(* IEC 61131-3 sources: AXOpen/src/components.festo.drives/ctrl/src/AxoCmmtAs, 11 files *)

(* ---- AxoCmmtAsErrorStruct.st ---- *)
NAMESPACE AXOpen.Components.Festo.Drives
    TYPE
        {S7.extern=ReadWrite}
        AxoCmmtAsErrorStruct :
        STRUCT
            Table       : AXOpen.Components.Festo.Drives.eAxoCmmtAsErrorTable;          (* Additional diagnosis table           *)
            Additional1 : DWORD;                (* Additional diagnosis number1         *)
            Additional2 : DWORD;                (* Additional diagnosis number2         *)
        END_STRUCT;
    END_TYPE
END_NAMESPACE

(* ---- eAxoCmmtAsErrorCode.st ---- *)
NAMESPACE AXOpen.Components.Festo.Drives
    TYPE PUBLIC
        eAxoCmmtAsErrorCode : WORD
        (
            NONE_ERROR                  := WORD#16#0000,     (* No error code available              *)
            (*                  invalid input                                                   *)
            INPUT_INVALID_ERROR         := WORD#16#0001,     (* Invalid input                        *)
            (*                  communications error                                            *)
            COMMUNICATION_ERROR         := WORD#16#0002,     (* Error while communication            *)
            (*                  data processing error                                           *)
            RESOURCE_ERROR              := WORD#16#0003,     (* Resource error                       *)
            ACCESS_ERROR                := WORD#16#0004,     (* Access error                         *)
            STATE_MACHINE_ERROR         := WORD#16#0005,     (* Invalid state State - Machine        *)
            INPUT_RANGE_ERROR           := WORD#16#0006,     (* Error because Input out of range     *)
            CALCULATION_ERROR           := WORD#16#0007,     (* Error while calculation              *)
            (*                  device error                                                    *)
            DEVICE_ERROR                := WORD#16#0008,     (* Device Error occurred                *)
            (*                  other error                                                     *)
            OTHER_ERROR                 := WORD#16#7FFE,     (* Undefined Error                      *)
            (*                  system error                                                    *)
            SYSTEM_ERROR                := WORD#16#7FFF      (* System error occured                 *)

                );
    END_TYPE
END_NAMESPACE

(* ---- eAxoCmmtAsErrorTable.st ---- *)
NAMESPACE AXOpen.Components.Festo.Drives
    TYPE PUBLIC
        eAxoCmmtAsErrorTable : WORD
        (
            NO_TABLE_USED           := WORD#16#0000,         //reserved
            SERCOS_TABLE            := WORD#16#0010,         //Sercos Error: Addtitional1 = Sercos Code
            MLDS_TABLE              := WORD#16#0020,         //Drive-based Motion - Logic
            MLC_TABLE               := WORD#16#0030,         //Controller - based Motion - Logic
            MTX_TABLE               := WORD#16#0040,         //CNC
            MLP_TABLE               := WORD#16#0050,         //PC  - based Motion Logic
            PLC_TABLE               := WORD#16#0060,         //PLC
            INDRV_TABLE             := WORD#16#0070,         //IndraDrive
            DIAX_TABLE              := WORD#16#0080,         //DIAX
            ECO_TABLE               := WORD#16#0090,         //EcoDrive
            PB_DP_TABLE             := WORD#16#0130,         //Profibus
            DEVICENET_TABLE         := WORD#16#0140,         //DeviceNet
            ETHERNET_TABLE          := WORD#16#0150,         //Ethernet
            INTERBUS_TABLE          := WORD#16#0160,         //Interbus
            F_RELATED_TABLE         := WORD#16#0170,         //function related
            USER1_TABLE             := WORD#16#1000,         //free User Table
            USER2_TABLE             := WORD#16#1001,         //free User Table
            USER3_TABLE             := WORD#16#1002,         //free User Table
            USER4_TABLE             := WORD#16#1003,         //free User Table
            USER5_TABLE             := WORD#16#1004,         //free User Table
            USER6_TABLE             := WORD#16#1005,         //free User Table
            USER7_TABLE             := WORD#16#1006,         //free User Table
            USER8_TABLE             := WORD#16#1007,         //free User Table
            USER9_TABLE             := WORD#16#1008,         //free User Table
            USER10_TABLE            := WORD#16#1009          //free User Table
        );
    END_TYPE
END_NAMESPACE

(* ---- AxoCmmtAs.st ---- *)
USING AXOpen.Components.Drives;
USING AXOpen.Core;
USING AXOpen.Messaging.Static;
USING AXOpen.Messaging;
USING AXOpen.Core;
USING AXOpen.Components.Abstractions;
USING AXOpen.Components.Abstractions.Drives;
USING AXOpen.Components.Drives;
USING System.Math;
USING System.BitAccess;
USING Siemens.Simatic.Hardware.Utilities;

NAMESPACE AXOpen.Components.Festo.Drives

    {#ix-attr:[Container(Layout.Wrap)]}
    {S7.extern=ReadWrite}
    CLASS PUBLIC AxoCmmtAs EXTENDS AXOpen.Components.Drives.AxoDrive IMPLEMENTS AXOpen.Components.Abstractions.Drives.IAxoDrive
        VAR PUBLIC //STATUS
            {#ix-attr:[Container(Layout.Stack)]}
            {#ix-attr:[ComponentDetails("Status")]}
            {#ix-attr:[ReadOnly()]}
            DriveStatus         :   AxoCmmtAs_Component_Status;
            Messenger           :   AXOpen.Messaging.Static.AxoMessenger;
            TaskMessenger       :   AXOpen.Messaging.Static.AxoMessenger;
        END_VAR
        VAR PUBLIC // HwDiag
            {#ix-attr:[Container(Layout.Stack)]}
            {#ix-attr:[ComponentDetails("Hardware diagnostics")]}
            {#ix-set:AttributeName = "<#Update diagnostics#>"}
            HardwareDiagnosticsTask :   AXOpen.Io.AxoHardwareDiagnostics;
        END_VAR
        VAR PUBLIC // AxisRef
            {#ix-attr:[Container(Layout.Stack)]}
            {#ix-attr:[ComponentDetails("AxisRef")]}
            {#ix-attr:[ReadOnly()]}
            AxisRefExt :  AXOpen.Components.Festo.Drives.AxoCmmtAsAxisReference;
        END_VAR
        VAR PUBLIC // Scaling
            {#ix-attr:[Container(Layout.Stack)]}
            {#ix-attr:[ComponentDetails("Scaling")]}
            {#ix-attr:[ReadOnly()]}
            {#ix-set:AttributeName = "<#Scaling constant required position#>"}
            {#ix-set:AttributeToolTip = "<#Depends on the actual settings in the Festo Automation Suite#>"}
            ScalingConstantRequiredPosition         :   LREAL   :=  1000;
            {#ix-attr:[ComponentDetails("Scaling")]}
            {#ix-attr:[ReadOnly()]}
            {#ix-set:AttributeName = "<#Scaling constant actual position#>"}
            {#ix-set:AttributeToolTip = "<#Depends on the actual settings in the Festo Automation Suite#>"}
            ScalingConstantActualPosition         :   LREAL   :=  0.001;
            {#ix-attr:[ComponentDetails("Scaling")]}
            {#ix-attr:[ReadOnly()]}
            {#ix-set:AttributeName = "<#Scaling constant required velocity#>"}
            {#ix-set:AttributeToolTip = "<#Depends on the actual settings in the Festo Automation Suite#>"}
            ScalingConstantRequiredVelocity         :   LREAL   :=  1;
            {#ix-attr:[ComponentDetails("Scaling")]}
            {#ix-attr:[ReadOnly()]}
            {#ix-set:AttributeName = "<#Scaling constant actual velocity#>"}
            {#ix-set:AttributeToolTip = "<#Depends on the actual settings in the Festo Automation Suite#>"}
            ScalingConstantActualVelocity         :   LREAL   :=  0.000000000931322574615478515625;
            {#ix-attr:[ComponentDetails("Scaling")]}
            {#ix-attr:[ReadOnly()]}
            {#ix-set:AttributeName = "<#Scaling constant required torque#>"}
            {#ix-set:AttributeToolTip = "<#Depends on the actual settings in the Festo Automation Suite#>"}
            ScalingConstantRequiredTorque         :   LREAL   :=  1;
            {#ix-attr:[ComponentDetails("Scaling")]}
            {#ix-attr:[ReadOnly()]}
            {#ix-set:AttributeName = "<#Scaling constant actual torque#>"}
            {#ix-set:AttributeToolTip = "<#Depends on the actual settings in the Festo Automation Suite#>"}
            ScalingConstantActualTorque         :   LREAL   :=  0.00006103515625;
            {#ix-attr:[ComponentDetails("Scaling")]}
            {#ix-attr:[ReadOnly()]}
            {#ix-set:AttributeName = "<#Scaling constant required acceleration#>"}
            {#ix-set:AttributeToolTip = "<#Depends on the actual settings in the Festo Automation Suite#>"}
            ScalingConstantRequiredAcceleration        :   LREAL   :=  LREAL#16.384;
            {#ix-attr:[ComponentDetails("Scaling")]}
            {#ix-attr:[ReadOnly()]}
            {#ix-set:AttributeName = "<#Scaling constant actual acceleration#>"}
            {#ix-set:AttributeToolTip = "<#Depends on the actual settings in the Festo Automation Suite#>"}
            ScalingConstantActualAcceleration        :   LREAL   :=  LREAL#0.06103515625;
            {#ix-attr:[ComponentDetails("Scaling")]}
            {#ix-attr:[ReadOnly()]}
            {#ix-set:AttributeName = "<#Scaling constant required deceleration#>"}
            {#ix-set:AttributeToolTip = "<#Depends on the actual settings in the Festo Automation Suite#>"}
            ScalingConstantRequiredDeceleration        :   LREAL   :=  LREAL#16.384;
            {#ix-attr:[ComponentDetails("Scaling")]}
            {#ix-attr:[ReadOnly()]}
            {#ix-set:AttributeName = "<#Scaling constant actual deceleration#>"}
            {#ix-set:AttributeToolTip = "<#Depends on the actual settings in the Festo Automation Suite#>"}
            ScalingConstantActualDeceleration        :   LREAL   :=  LREAL#0.06103515625;
            {#ix-attr:[ComponentDetails("Scaling")]}
            {#ix-attr:[ReadOnly()]}
            {#ix-set:AttributeName = "<#Scaling constant required jerk#>"}
            {#ix-set:AttributeToolTip = "<#Depends on the actual settings in the Festo Automation Suite#>"}
            ScalingConstantRequiredJerk        :   LREAL   :=  LREAL#0.001;
            {#ix-attr:[ComponentDetails("Scaling")]}
            {#ix-attr:[ReadOnly()]}
            {#ix-set:AttributeName = "<#Scaling constant actual jerk#>"}
            {#ix-set:AttributeToolTip = "<#Depends on the actual settings in the Festo Automation Suite#>"}
            ScalingConstantActualJerk        :   LREAL   :=  LREAL#1000.0;
            {#ix-attr:[ComponentDetails("Scaling")]}
            {#ix-attr:[ReadOnly()]}
            {#ix-set:AttributeName = "<#Axis type#>"}
            {#ix-set:AttributeToolTip = "<#Depends on the actual settings in the Festo Automation Suite#>"}
            AxisType    :   eAxoDriveAxisType := eAxoDriveAxisType#Undefined;
        END_VAR

        VAR PUBLIC //   Debug
            {#ix-attr:[Container(Layout.Stack)]}
            {#ix-attr:[ComponentHeader()]}
            State : UINT;
            {#ix-attr:[Container(Layout.Stack)]}
            {#ix-attr:[ComponentHeader()]}
            ScalingReadState : UINT;
            {#ix-attr:[Container(Layout.Stack)]}
            {#ix-attr:[ComponentHeader()]}
            Debug : LINT;
        END_VAR

        VAR PRIVATE
            _ScalingRead            :   BOOL := FALSE;
            PNU_11724               :   LINT;       //  Resolution position (P1.7841.0.0)
            PNU_11725               :   LINT;       //  Resolution velocity (P1.7842.0.0)
            PNU_11726               :   LINT;       //  Resolution acceleration (P1.7843.0.0)
            PNU_11727               :   LINT;       //  Resolution jerk (P1.7844.0.0)
            PNU_12345               :   REAL;       //  Base value velocity (P1.11280701.0.0)
            PNU_11122               :   REAL;       //  Maximum motor torque/servo drive (P1.381.0.0)
            PNU_810                 :   REAL;       //  Base value acceleration (P1.11280702.0.0)
            PNU_811                 :   REAL;       //  Base value deceleration (P1.11280703.0.0)
            PNU_11203               :   BOOL;       //  Move to axis zero point after homing (P1.841.0.0)
            PNU_11734               :   LINT;       //  Axis zero point offset (P1.8416.0.0)
            PNU_11735               :   LINT;       //  Referencing method (P1.8417.0.0)
            PNU_12694               :   LINT;       //  User unit position (P1.7851.0.0)
            PNU_12695               :   LINT;       //  User unit velocity (P1.7852.0.0)
            PNU_12696               :   LINT;       //  User unit acceleration (P1.7853.0.0)
            PNU_12697               :   LINT;       //  User unit jerk (P1.7854.0.0)

            Parametrization         :   AxoReadWritePROFIdriveParameter;

            _initHwCheckDone        :   BOOL;
            _retval                 :   WORD;
            _geoAddr                :   GeoAddr;
            _outHwid                :   UINT;
            _blink                  :   AXOpen.Timers.AxoBlinker;
            _inputsAddress          :   UDINT;
            _inputsCount            :   UINT;
            _outputsAddress         :   UDINT;
            _outputsCount           :   UINT;
            _infoTimer              :   AXOpen.Timers.OnDelayTimer;
            _errorTimer             :   AXOpen.Timers.OnDelayTimer;
            _scalingReadState       :   UINT;

        END_VAR

        ///<summary>
        /// Runs tasks and logic of this component.
        /// >[!IMPORTANT] This method or one of its overloads must be called cyclically.
        ///</summary>
        METHOD PUBLIC Run
            VAR_INPUT
                inParent            :   IAxoObject;
                hwID                :   UINT;
                Enable              :   BOOL;                       //  As long as ‘Enable’ is true, power is being enabled.
                EnablePositive      :   BOOL;                       //  As long as ‘Enable’ is true, this permits motion in positive direction
                EnableNegative      :   BOOL;                       //  As long as ‘Enable’ is true, this permits motion in negative direction
            END_VAR
            VAR
                // _AxisReference  :   REF_TO AXOpen.Components.Festo.Drives.AxoCmmtAsAxisReference;
                tempDWord       :   DWORD;
                //                                      |     -10   |     -9    |    -8    |    -7   |   -6   |   -5  |  -4  | -3  | -2 |-1|  0 | 1  |  2  |  3   |   4   |   5    |   6     |    7     |     8     |    9      |     10    |
                _exp    :   ARRAY [-10..10] OF LREAL := [0.000000001,0.000000001,0.00000001,0.0000001,0.000001,0.00001,0.0001,0.001,0.01,0.1,1.0,10.0,100.0,1000.0,10000.0,100000.0,1000000.0,10000000.0,100000000.0,100000000.0,100000000.0];
            END_VAR
            SUPER.Run(inParent);
            Messenger.Serve(THIS);

            ScalingReadState       :=  _scalingReadState;

            IF NOT _initHwCheckDone THEN
                IF inParent = NULL THEN
                    Messenger.Activate(     UINT#700, eAxoMessageCategory#ProgrammingError);
                    DriveStatus.Error.Id := UINT#700;
                    RETURN;
                END_IF;
                AxisRefExt.HWIDs.HW_Device  :=  hwID;
                IF AxisRefExt.HWIDs.HW_Device = UINT#0 THEN
                    Messenger.Activate(     UINT#701, eAxoMessageCategory#ProgrammingError);
                    DriveStatus.Error.Id := UINT#701;
                    RETURN;
                END_IF;

                _retval := ReadSlotFromHardwareID(hardwareID := AxisRefExt.HWIDs.HW_Device, geoAddr :=_geoAddr);
                IF _retval = WORD#8090 THEN
                    Messenger.Activate(     UINT#702,eAxoMessageCategory#Error);
                    DriveStatus.Error.Id := UINT#702;
                    RETURN;
                END_IF;

                //******************Slot 1*****************//
                _geoAddr.Slot   :=  UINT#1;
                _geoAddr.HardwareType := UINT#4; // (4-Module)
                _retval := ReadHardwareIDFromSlot(geoAddr := _geoAddr, hardwareID => AxisRefExt.HWIDs.HW_DoServo);
                IF AxisRefExt.HWIDs.HW_DoServo = UINT#0 THEN
                    Messenger.Activate(     UINT#710,eAxoMessageCategory#Error);
                    DriveStatus.Error.Id := UINT#710;
                    RETURN;
                END_IF;
                IF _retval = WORD#8091 THEN
                    Messenger.Activate(     UINT#711,eAxoMessageCategory#Error);
                    DriveStatus.Error.Id := UINT#711;
                    RETURN;
                END_IF;
                IF _retval = WORD#8094 THEN
                    Messenger.Activate(     UINT#712,eAxoMessageCategory#Error);
                    DriveStatus.Error.Id := UINT#712;
                    RETURN;
                END_IF;
                IF _retval = WORD#8095 THEN
                    Messenger.Activate(     UINT#713,eAxoMessageCategory#Error);
                    DriveStatus.Error.Id := UINT#713;
                    RETURN;
                END_IF;
                IF _retval = WORD#8096 THEN
                    Messenger.Activate(     UINT#714,eAxoMessageCategory#Error);
                    DriveStatus.Error.Id := UINT#714;
                    RETURN;
                END_IF;
                IF _retval = WORD#8097 THEN
                    Messenger.Activate(     UINT#715,eAxoMessageCategory#Error);
                    DriveStatus.Error.Id := UINT#715;
                    RETURN;
                END_IF;
                ReadHardwareIOAddress(hardwareID := (AxisRefExt.HWIDs.HW_DoServo) , inputStartAddress => _inputsAddress , inputCount => _inputsCount , outputStartAddress => _outputsAddress , outputCount => _outputsCount);
                IF _inputsCount <> UINT#0 OR _outputsCount <> UINT#0 THEN
                    Messenger.Activate(     UINT#716,eAxoMessageCategory#Error);
                    DriveStatus.Error.Id := UINT#716;
                    RETURN;
                END_IF;
                //******************Slot 1*****************//
                _geoAddr.Slot   :=  UINT#1;
                //******************Subslot 0**************//
                _geoAddr.Subslot   :=  UINT#0;
                _geoAddr.HardwareType := UINT#5; // (5-Submodule)
                _retval := ReadHardwareIDFromSlot(geoAddr := _geoAddr, hardwareID => AxisRefExt.HWIDs.HW_DoServoSub);
                IF AxisRefExt.HWIDs.HW_DoServoSub = UINT#0 THEN
                    Messenger.Activate(     UINT#720,eAxoMessageCategory#Error);
                    DriveStatus.Error.Id := UINT#720;
                    RETURN;
                END_IF;
                IF _retval = WORD#8091 THEN
                    Messenger.Activate(     UINT#721,eAxoMessageCategory#Error);
                    DriveStatus.Error.Id := UINT#721;
                    RETURN;
                END_IF;
                IF _retval = WORD#8094 THEN
                    Messenger.Activate(     UINT#722,eAxoMessageCategory#Error);
                    DriveStatus.Error.Id := UINT#722;
                    RETURN;
                END_IF;
                IF _retval = WORD#8095 THEN
                    Messenger.Activate(     UINT#723,eAxoMessageCategory#Error);
                    DriveStatus.Error.Id := UINT#723;
                    RETURN;
                END_IF;
                IF _retval = WORD#8096 THEN
                    Messenger.Activate(     UINT#724,eAxoMessageCategory#Error);
                    DriveStatus.Error.Id := UINT#724;
                    RETURN;
                END_IF;
                IF _retval = WORD#8097 THEN
                    Messenger.Activate(     UINT#725,eAxoMessageCategory#Error);
                    DriveStatus.Error.Id := UINT#725;
                    RETURN;
                END_IF;
                ReadHardwareIOAddress(hardwareID := (AxisRefExt.HWIDs.HW_DoServoSub) , inputStartAddress => _inputsAddress , inputCount => _inputsCount , outputStartAddress => _outputsAddress , outputCount => _outputsCount);
                IF _inputsCount <> UINT#0 OR _outputsCount <> UINT#0 THEN
                    Messenger.Activate(     UINT#726,eAxoMessageCategory#Error);
                    DriveStatus.Error.Id := UINT#726;
                    RETURN;
                END_IF;
                //******************Slot 1*****************//
                _geoAddr.Slot   :=  UINT#1;
                //******************Subslot 1**************//
                _geoAddr.Subslot   :=  UINT#1;
                _geoAddr.HardwareType := UINT#5; // (5-Submodule)
                _retval := ReadHardwareIDFromSlot(geoAddr := _geoAddr, hardwareID => AxisRefExt.HWIDs.HW_ModuleAccessPoint);
                IF AxisRefExt.HWIDs.HW_ModuleAccessPoint = UINT#0 THEN
                    Messenger.Activate(     UINT#730,eAxoMessageCategory#Error);
                    DriveStatus.Error.Id := UINT#730;
                    RETURN;
                END_IF;
                IF _retval = WORD#8091 THEN
                    Messenger.Activate(     UINT#731,eAxoMessageCategory#Error);
                    DriveStatus.Error.Id := UINT#731;
                    RETURN;
                END_IF;
                IF _retval = WORD#8094 THEN
                    Messenger.Activate(     UINT#732,eAxoMessageCategory#Error);
                    DriveStatus.Error.Id := UINT#732;
                    RETURN;
                END_IF;
                IF _retval = WORD#8095 THEN
                    Messenger.Activate(     UINT#733,eAxoMessageCategory#Error);
                    DriveStatus.Error.Id := UINT#733;
                    RETURN;
                END_IF;
                IF _retval = WORD#8096 THEN
                    Messenger.Activate(     UINT#734,eAxoMessageCategory#Error);
                    DriveStatus.Error.Id := UINT#734;
                    RETURN;
                END_IF;
                IF _retval = WORD#8097 THEN
                    Messenger.Activate(     UINT#735,eAxoMessageCategory#Error);
                    DriveStatus.Error.Id := UINT#735;
                    RETURN;
                END_IF;
                ReadHardwareIOAddress(hardwareID := (AxisRefExt.HWIDs.HW_ModuleAccessPoint) , inputStartAddress => _inputsAddress , inputCount => _inputsCount , outputStartAddress => _outputsAddress , outputCount => _outputsCount);
                IF _inputsCount <> UINT#0 OR _outputsCount <> UINT#0 THEN
                    Messenger.Activate(     UINT#736,eAxoMessageCategory#Error);
                    DriveStatus.Error.Id := UINT#736;
                    RETURN;
                END_IF;
                //******************Slot 1*****************//
                _geoAddr.Slot   :=  UINT#1;
                //******************Subslot 2**************//
                _geoAddr.Subslot   :=  UINT#2;
                _geoAddr.HardwareType := UINT#5; // (5-Submodule)
                _retval := ReadHardwareIDFromSlot(geoAddr := _geoAddr, hardwareID => AxisRefExt.HWIDs.HW_EmptyModule_1);
                IF AxisRefExt.HWIDs.HW_EmptyModule_1 = UINT#0 THEN
                    Messenger.Activate(     UINT#740,eAxoMessageCategory#Error);
                    DriveStatus.Error.Id := UINT#740;
                    RETURN;
                END_IF;
                IF _retval = WORD#8091 THEN
                    Messenger.Activate(     UINT#741,eAxoMessageCategory#Error);
                    DriveStatus.Error.Id := UINT#741;
                    RETURN;
                END_IF;
                IF _retval = WORD#8094 THEN
                    Messenger.Activate(     UINT#742,eAxoMessageCategory#Error);
                    DriveStatus.Error.Id := UINT#742;
                    RETURN;
                END_IF;
                IF _retval = WORD#8095 THEN
                    Messenger.Activate(     UINT#743,eAxoMessageCategory#Error);
                    DriveStatus.Error.Id := UINT#743;
                    RETURN;
                END_IF;
                IF _retval = WORD#8096 THEN
                    Messenger.Activate(     UINT#744,eAxoMessageCategory#Error);
                    DriveStatus.Error.Id := UINT#744;
                    RETURN;
                END_IF;
                IF _retval = WORD#8097 THEN
                    Messenger.Activate(     UINT#745,eAxoMessageCategory#Error);
                    DriveStatus.Error.Id := UINT#745;
                    RETURN;
                END_IF;
                ReadHardwareIOAddress(hardwareID := (AxisRefExt.HWIDs.HW_EmptyModule_1) , inputStartAddress => _inputsAddress , inputCount => _inputsCount , outputStartAddress => _outputsAddress , outputCount => _outputsCount);
                IF _inputsCount <> UINT#0 OR _outputsCount <> UINT#0 THEN
                    Messenger.Activate(     UINT#746,eAxoMessageCategory#Error);
                    DriveStatus.Error.Id := UINT#746;
                    RETURN;
                END_IF;
                //******************Slot 1*****************//
                _geoAddr.Slot   :=  UINT#1;
                //******************Subslot 3**************//
                _geoAddr.Subslot   :=  UINT#3;
                _geoAddr.HardwareType := UINT#5; // (5-Submodule)
                _retval := ReadHardwareIDFromSlot(geoAddr := _geoAddr, hardwareID => AxisRefExt.HWIDs.HW_Telegram111);
                IF AxisRefExt.HWIDs.HW_Telegram111 = UINT#0 THEN
                    Messenger.Activate(     UINT#750,eAxoMessageCategory#Error);
                    DriveStatus.Error.Id := UINT#750;
                    RETURN;
                END_IF;
                IF _retval = WORD#8091 THEN
                    Messenger.Activate(     UINT#751,eAxoMessageCategory#Error);
                    DriveStatus.Error.Id := UINT#751;
                    RETURN;
                END_IF;
                IF _retval = WORD#8094 THEN
                    Messenger.Activate(     UINT#752,eAxoMessageCategory#Error);
                    DriveStatus.Error.Id := UINT#752;
                    RETURN;
                END_IF;
                IF _retval = WORD#8095 THEN
                    Messenger.Activate(     UINT#753,eAxoMessageCategory#Error);
                    DriveStatus.Error.Id := UINT#753;
                    RETURN;
                END_IF;
                IF _retval = WORD#8096 THEN
                    Messenger.Activate(     UINT#754,eAxoMessageCategory#Error);
                    DriveStatus.Error.Id := UINT#754;
                    RETURN;
                END_IF;
                IF _retval = WORD#8097 THEN
                    Messenger.Activate(     UINT#755,eAxoMessageCategory#Error);
                    DriveStatus.Error.Id := UINT#755;
                    RETURN;
                END_IF;
                ReadHardwareIOAddress(hardwareID := (AxisRefExt.HWIDs.HW_Telegram111) , inputStartAddress => _inputsAddress , inputCount => _inputsCount , outputStartAddress => _outputsAddress , outputCount => _outputsCount);
                IF _inputsCount <> UINT#24 OR _outputsCount <> UINT#24 THEN
                    Messenger.Activate(     UINT#756,eAxoMessageCategory#Error);
                    DriveStatus.Error.Id := UINT#756;
                    RETURN;
                END_IF;
                //******************Slot 1*****************//
                _geoAddr.Slot   :=  UINT#1;
                //******************Subslot 4**************//
                _geoAddr.Subslot   :=  UINT#4;
                _geoAddr.HardwareType := UINT#5; // (5-Submodule)
                _retval := ReadHardwareIDFromSlot(geoAddr := _geoAddr, hardwareID => AxisRefExt.HWIDs.HW_EmptyModule_2);
                IF AxisRefExt.HWIDs.HW_EmptyModule_2 = UINT#0 THEN
                    Messenger.Activate(     UINT#760,eAxoMessageCategory#Error);
                    DriveStatus.Error.Id := UINT#760;
                    RETURN;
                END_IF;
                IF _retval = WORD#8091 THEN
                    Messenger.Activate(     UINT#761,eAxoMessageCategory#Error);
                    DriveStatus.Error.Id := UINT#761;
                    RETURN;
                END_IF;
                IF _retval = WORD#8094 THEN
                    Messenger.Activate(     UINT#762,eAxoMessageCategory#Error);
                    DriveStatus.Error.Id := UINT#762;
                    RETURN;
                END_IF;
                IF _retval = WORD#8095 THEN
                    Messenger.Activate(     UINT#763,eAxoMessageCategory#Error);
                    DriveStatus.Error.Id := UINT#763;
                    RETURN;
                END_IF;
                IF _retval = WORD#8096 THEN
                    Messenger.Activate(     UINT#764,eAxoMessageCategory#Error);
                    DriveStatus.Error.Id := UINT#764;
                    RETURN;
                END_IF;
                IF _retval = WORD#8097 THEN
                    Messenger.Activate(     UINT#765,eAxoMessageCategory#Error);
                    DriveStatus.Error.Id := UINT#765;
                    RETURN;
                END_IF;
                ReadHardwareIOAddress(hardwareID := (AxisRefExt.HWIDs.HW_EmptyModule_2) , inputStartAddress => _inputsAddress , inputCount => _inputsCount , outputStartAddress => _outputsAddress , outputCount => _outputsCount);
                IF _inputsCount <> UINT#0 OR _outputsCount <> UINT#0 THEN
                    Messenger.Activate(     UINT#766,eAxoMessageCategory#Error);
                    DriveStatus.Error.Id := UINT#766;
                    RETURN;
                END_IF;
                //******************Slot 1*****************//
                _geoAddr.Slot   :=  UINT#1;
                //******************Subslot 5**************//
                _geoAddr.Subslot   :=  UINT#5;
                _geoAddr.HardwareType := UINT#5; // (5-Submodule)
                _retval := ReadHardwareIDFromSlot(geoAddr := _geoAddr, hardwareID => AxisRefExt.HWIDs.HW_Telegram750);
                IF AxisRefExt.HWIDs.HW_Telegram750 = UINT#0 THEN
                    Messenger.Activate(     UINT#770,eAxoMessageCategory#Error);
                    DriveStatus.Error.Id := UINT#770;
                    RETURN;
                END_IF;
                IF _retval = WORD#8091 THEN
                    Messenger.Activate(     UINT#771,eAxoMessageCategory#Error);
                    DriveStatus.Error.Id := UINT#771;
                    RETURN;
                END_IF;
                IF _retval = WORD#8094 THEN
                    Messenger.Activate(     UINT#772,eAxoMessageCategory#Error);
                    DriveStatus.Error.Id := UINT#772;
                    RETURN;
                END_IF;
                IF _retval = WORD#8095 THEN
                    Messenger.Activate(     UINT#773,eAxoMessageCategory#Error);
                    DriveStatus.Error.Id := UINT#773;
                    RETURN;
                END_IF;
                IF _retval = WORD#8096 THEN
                    Messenger.Activate(     UINT#774,eAxoMessageCategory#Error);
                    DriveStatus.Error.Id := UINT#774;
                    RETURN;
                END_IF;
                IF _retval = WORD#8097 THEN
                    Messenger.Activate(     UINT#775,eAxoMessageCategory#Error);
                    DriveStatus.Error.Id := UINT#775;
                    RETURN;
                END_IF;
                ReadHardwareIOAddress(hardwareID := (AxisRefExt.HWIDs.HW_Telegram750) , inputStartAddress => _inputsAddress , inputCount => _inputsCount , outputStartAddress => _outputsAddress , outputCount => _outputsCount);
                IF _inputsCount <> UINT#2 OR _outputsCount <> UINT#8 THEN
                    Messenger.Activate(     UINT#776,eAxoMessageCategory#Error);
                    DriveStatus.Error.Id := UINT#776;
                    RETURN;
                END_IF;
                // *********************************************

                IF inParent = NULL THEN
                    Messenger.Activate(     UINT#1130,eAxoMessageCategory#Error);
                    DriveStatus.Error.Id := UINT#1130;
                    RETURN;
                END_IF;
                IF  AxisRefExt.HWIDs.HW_Device = UINT#0 THEN
                    Messenger.Activate(     UINT#1131,eAxoMessageCategory#Error);
                    DriveStatus.Error.Id := UINT#1131;
                    RETURN;
                END_IF;

                IF AxisRefExt.HWIDs.HW_DoServo  = UINT#0 THEN
                    Messenger.Activate(     UINT#1132,eAxoMessageCategory#Error);
                    DriveStatus.Error.Id := UINT#1132;
                    RETURN;
                END_IF;
                IF AxisRefExt.HWIDs.HW_ModuleAccessPoint  = UINT#0 THEN
                    Messenger.Activate(     UINT#1133,eAxoMessageCategory#Error);
                    DriveStatus.Error.Id := UINT#1133;
                    RETURN;
                END_IF;
                IF AxisRefExt.HWIDs.HW_EmptyModule_1 = UINT#0 THEN
                    Messenger.Activate(     UINT#1134,eAxoMessageCategory#Error);
                    DriveStatus.Error.Id := UINT#1134;
                    RETURN;
                END_IF;
                IF AxisRefExt.HWIDs.HW_Telegram111 = UINT#0 THEN
                    Messenger.Activate(     UINT#1135,eAxoMessageCategory#Error);
                    DriveStatus.Error.Id := UINT#1135;
                    RETURN;
                END_IF;
                IF AxisRefExt.HWIDs.HW_EmptyModule_2   = UINT#0 THEN
                    Messenger.Activate(     UINT#1136,eAxoMessageCategory#Error);
                    DriveStatus.Error.Id := UINT#1136;
                    RETURN;
                END_IF;
                IF AxisRefExt.HWIDs.HW_Telegram750  = UINT#0 THEN
                    Messenger.Activate(     UINT#1137,eAxoMessageCategory#Error);
                    DriveStatus.Error.Id := UINT#1137;
                    RETURN;
                END_IF;

                _initHwCheckDone    := TRUE;
            END_IF;
            Messenger.ActivateOnCondition(ULINT#1800, NOT _ScalingRead, eAxoMessageCategory#Potential);
            //********************Diagnostics******************//
            HardwareDiagnosticsTask.Run(THIS,AxisRefExt.HWIDs.HW_Device);
            //********************PARAMETRIZAION***************//
            Parametrization.Run(THIS);
            Parametrization.Inputs.HardwareId := AxisRefExt.HWIDs.HW_ModuleAccessPoint;
            //*******************SCALING***********************//
            IF NOT _ScalingRead THEN
                Messenger.Activate(ULINT#1800 , eAxoMessageCategory#Potential);
                IF _scalingReadState = UINT#0 THEN
                    AxisType := eAxoDriveAxisType#Undefined;
                    _scalingReadState := UINT#1;
                    State := UINT#1;
                END_IF;
                //Reading PNU 11724 Factor group Position
                IF _scalingReadState = UINT#1 THEN
                    Parametrization.Inputs.Enable := TRUE;
                    Parametrization.Inputs.ReadWrite   := FALSE;
                    Parametrization.Inputs.ParameterNo := 11724;
                    Parametrization.Inputs.Subindex    := 0;
                    Parametrization.Inputs.AxisNo  := BYTE#1;
                    Parametrization.Inputs.HardwareId  := AxisRefExt.HWIDs.HW_ModuleAccessPoint;
                    IF Parametrization.Outputs.Done AND NOT Parametrization.Outputs.Error THEN
                        PNU_11724 := Parametrization.Outputs.ValueReadLINT;
                        _scalingReadState := UINT#2;
                    END_IF;
                END_IF;
                IF _scalingReadState = UINT#2 THEN
                    Parametrization.Inputs.Enable := FALSE;
                    IF NOT Parametrization.Outputs.Done THEN
                        _scalingReadState := UINT#3;
                    END_IF;
                END_IF;
                //Reading PNU 11725 Factor group Velocity
                IF _scalingReadState = UINT#3 THEN
                    Parametrization.Inputs.Enable := TRUE;
                    Parametrization.Inputs.ReadWrite   := FALSE;
                    Parametrization.Inputs.ParameterNo := 11725;
                    Parametrization.Inputs.Subindex    := 0;
                    Parametrization.Inputs.AxisNo  := BYTE#1;
                    Parametrization.Inputs.HardwareId  := AxisRefExt.HWIDs.HW_ModuleAccessPoint;
                    IF Parametrization.Outputs.Done AND NOT Parametrization.Outputs.Error THEN
                        PNU_11725 := Parametrization.Outputs.ValueReadLINT;
                        _scalingReadState := UINT#4;
                    END_IF;
                END_IF;
                IF _scalingReadState = UINT#4 THEN
                    Parametrization.Inputs.Enable := FALSE;
                    IF NOT Parametrization.Outputs.Done THEN
                        _scalingReadState := UINT#5;
                    END_IF;
                END_IF;
                //Reading PNU 12345 Base value velocity
                IF _scalingReadState = UINT#5 THEN
                    Parametrization.Inputs.Enable := TRUE;
                    Parametrization.Inputs.ReadWrite   := FALSE;
                    Parametrization.Inputs.ParameterNo := 12345;
                    Parametrization.Inputs.Subindex    := 0;
                    Parametrization.Inputs.AxisNo  := BYTE#1;
                    Parametrization.Inputs.HardwareId  := AxisRefExt.HWIDs.HW_ModuleAccessPoint;
                    IF Parametrization.Outputs.Done AND NOT Parametrization.Outputs.Error THEN
                        PNU_12345 := Parametrization.Outputs.ValueReadREAL;
                        _scalingReadState := UINT#6;
                    END_IF;
                END_IF;
                IF _scalingReadState = UINT#6 THEN
                    Parametrization.Inputs.Enable := FALSE;
                    IF NOT Parametrization.Outputs.Done THEN
                        _scalingReadState := UINT#7;
                    END_IF;
                END_IF;
                //Reading PNU 11122 Maximum motor torque/servo drive
                IF _scalingReadState = UINT#7 THEN
                    Parametrization.Inputs.Enable := TRUE;
                    Parametrization.Inputs.ReadWrite   := FALSE;
                    Parametrization.Inputs.ParameterNo := 11122;
                    Parametrization.Inputs.Subindex    := 0;
                    Parametrization.Inputs.AxisNo  := BYTE#1;
                    Parametrization.Inputs.HardwareId  := AxisRefExt.HWIDs.HW_ModuleAccessPoint;
                    IF Parametrization.Outputs.Done AND NOT Parametrization.Outputs.Error THEN
                        PNU_11122 := Parametrization.Outputs.ValueReadREAL;
                        _scalingReadState := UINT#8;
                    END_IF;
                END_IF;
                IF _scalingReadState = UINT#8 THEN
                    Parametrization.Inputs.Enable := FALSE;
                    IF NOT Parametrization.Outputs.Done THEN
                        _scalingReadState := UINT#9;
                    END_IF;
                END_IF;
                //Reading PNU 810 Base value acceleration
                IF _scalingReadState = UINT#9 THEN
                    Parametrization.Inputs.Enable := TRUE;
                    Parametrization.Inputs.ReadWrite   := FALSE;
                    Parametrization.Inputs.ParameterNo := 810;
                    Parametrization.Inputs.Subindex    := 0;
                    Parametrization.Inputs.AxisNo  := BYTE#1;
                    Parametrization.Inputs.HardwareId  := AxisRefExt.HWIDs.HW_ModuleAccessPoint;
                    IF Parametrization.Outputs.Done AND NOT Parametrization.Outputs.Error THEN
                        PNU_810 := Parametrization.Outputs.ValueReadREAL;
                        _scalingReadState := UINT#10;
                    END_IF;
                END_IF;
                IF _scalingReadState = UINT#10 THEN
                    Parametrization.Inputs.Enable := FALSE;
                    IF NOT Parametrization.Outputs.Done THEN
                        _scalingReadState := UINT#11;
                    END_IF;
                END_IF;
                //Reading PNU 811 Base value deceleration
                IF _scalingReadState = UINT#11 THEN
                    Parametrization.Inputs.Enable := TRUE;
                    Parametrization.Inputs.ReadWrite   := FALSE;
                    Parametrization.Inputs.ParameterNo := 811;
                    Parametrization.Inputs.Subindex    := 0;
                    Parametrization.Inputs.AxisNo  := BYTE#1;
                    Parametrization.Inputs.HardwareId  := AxisRefExt.HWIDs.HW_ModuleAccessPoint;
                    IF Parametrization.Outputs.Done AND NOT Parametrization.Outputs.Error THEN
                        PNU_811 := Parametrization.Outputs.ValueReadREAL;
                        _scalingReadState := UINT#12;
                    END_IF;
                END_IF;
                IF _scalingReadState = UINT#12 THEN
                    Parametrization.Inputs.Enable := FALSE;
                    IF NOT Parametrization.Outputs.Done THEN
                        _scalingReadState := UINT#13;
                    END_IF;
                END_IF;
                //Reading PNU 11726 Resolution acceleration (P1.7843.0.0)
                IF _scalingReadState = UINT#13 THEN
                    Parametrization.Inputs.Enable := TRUE;
                    Parametrization.Inputs.ReadWrite   := FALSE;
                    Parametrization.Inputs.ParameterNo := 11726;
                    Parametrization.Inputs.Subindex    := 0;
                    Parametrization.Inputs.AxisNo  := BYTE#1;
                    Parametrization.Inputs.HardwareId  := AxisRefExt.HWIDs.HW_ModuleAccessPoint;
                    IF Parametrization.Outputs.Done AND NOT Parametrization.Outputs.Error THEN
                        PNU_11726 := Parametrization.Outputs.ValueReadLINT;
                        _scalingReadState := UINT#14;
                    END_IF;
                END_IF;
                IF _scalingReadState = UINT#14 THEN
                    Parametrization.Inputs.Enable := FALSE;
                    IF NOT Parametrization.Outputs.Done THEN
                        _scalingReadState := UINT#15;
                    END_IF;
                END_IF;
                //Reading PNU 11727 Resolution jerk (P1.7844.0.0)
                IF _scalingReadState = UINT#15 THEN
                    Parametrization.Inputs.Enable := TRUE;
                    Parametrization.Inputs.ReadWrite   := FALSE;
                    Parametrization.Inputs.ParameterNo := 11727;
                    Parametrization.Inputs.Subindex    := 0;
                    Parametrization.Inputs.AxisNo  := BYTE#1;
                    Parametrization.Inputs.HardwareId  := AxisRefExt.HWIDs.HW_ModuleAccessPoint;
                    IF Parametrization.Outputs.Done AND NOT Parametrization.Outputs.Error THEN
                        PNU_11727 := Parametrization.Outputs.ValueReadLINT;
                        _scalingReadState := UINT#16;
                    END_IF;
                END_IF;
                IF _scalingReadState = UINT#16 THEN
                    Parametrization.Inputs.Enable := FALSE;
                    IF NOT Parametrization.Outputs.Done THEN
                        _scalingReadState := UINT#17;
                    END_IF;
                END_IF;
                //Reading PNU PNU 12694 User unit position (P1.7851.0.0)
                IF _scalingReadState = UINT#17 THEN
                    Parametrization.Inputs.Enable := TRUE;
                    Parametrization.Inputs.ReadWrite   := FALSE;
                    Parametrization.Inputs.ParameterNo := 12694;
                    Parametrization.Inputs.Subindex    := 0;
                    Parametrization.Inputs.AxisNo  := BYTE#1;
                    Parametrization.Inputs.HardwareId  := AxisRefExt.HWIDs.HW_ModuleAccessPoint;
                    IF Parametrization.Outputs.Done AND NOT Parametrization.Outputs.Error THEN
                        PNU_12694 := Parametrization.Outputs.ValueReadLINT;
                        _scalingReadState := UINT#18;
                    END_IF;
                END_IF;
                IF _scalingReadState = UINT#18 THEN
                    Parametrization.Inputs.Enable := FALSE;
                    IF NOT Parametrization.Outputs.Done THEN
                        _scalingReadState := UINT#19;
                    END_IF;
                END_IF;
                //Reading PNU PNU 12695 User unit velocity (P1.7852.0.0)
                IF _scalingReadState = UINT#19 THEN
                    Parametrization.Inputs.Enable := TRUE;
                    Parametrization.Inputs.ReadWrite   := FALSE;
                    Parametrization.Inputs.ParameterNo := 12695;
                    Parametrization.Inputs.Subindex    := 0;
                    Parametrization.Inputs.AxisNo  := BYTE#1;
                    Parametrization.Inputs.HardwareId  := AxisRefExt.HWIDs.HW_ModuleAccessPoint;
                    IF Parametrization.Outputs.Done AND NOT Parametrization.Outputs.Error THEN
                        PNU_12695 := Parametrization.Outputs.ValueReadLINT;
                        _scalingReadState := UINT#20;
                    END_IF;
                END_IF;
                IF _scalingReadState = UINT#20 THEN
                    Parametrization.Inputs.Enable := FALSE;
                    IF NOT Parametrization.Outputs.Done THEN
                        _scalingReadState := UINT#21;
                    END_IF;
                END_IF;
                //Reading PNU PNU 12696 User unit acceleration (P1.7853.0.0)
                IF _scalingReadState = UINT#21 THEN
                    Parametrization.Inputs.Enable := TRUE;
                    Parametrization.Inputs.ReadWrite   := FALSE;
                    Parametrization.Inputs.ParameterNo := 12696;
                    Parametrization.Inputs.Subindex    := 0;
                    Parametrization.Inputs.AxisNo  := BYTE#1;
                    Parametrization.Inputs.HardwareId  := AxisRefExt.HWIDs.HW_ModuleAccessPoint;
                    IF Parametrization.Outputs.Done AND NOT Parametrization.Outputs.Error THEN
                        PNU_12696 := Parametrization.Outputs.ValueReadLINT;
                        _scalingReadState := UINT#22;
                    END_IF;
                END_IF;
                IF _scalingReadState = UINT#22 THEN
                    Parametrization.Inputs.Enable := FALSE;
                    IF NOT Parametrization.Outputs.Done THEN
                        _scalingReadState := UINT#23;
                    END_IF;
                END_IF;
                //Reading PNU PNU 12697 User unit jerk (P1.7854.0.0)
                IF _scalingReadState = UINT#23 THEN
                    Parametrization.Inputs.Enable := TRUE;
                    Parametrization.Inputs.ReadWrite   := FALSE;
                    Parametrization.Inputs.ParameterNo := 12697;
                    Parametrization.Inputs.Subindex    := 0;
                    Parametrization.Inputs.AxisNo  := BYTE#1;
                    Parametrization.Inputs.HardwareId  := AxisRefExt.HWIDs.HW_ModuleAccessPoint;
                    IF Parametrization.Outputs.Done AND NOT Parametrization.Outputs.Error THEN
                        PNU_12697 := Parametrization.Outputs.ValueReadLINT;
                        _scalingReadState := UINT#24;
                    END_IF;
                END_IF;
                IF _scalingReadState = UINT#24 THEN
                    Parametrization.Inputs.Enable := FALSE;
                    IF NOT Parametrization.Outputs.Done THEN
                        _scalingReadState := UINT#25;
                    END_IF;
                END_IF;
                //Check setting PNU 12694-12697 User unit position, velocity, acceleration and jerk are read correctly or not. If not, scaling will be wrong, so set the flag to FALSE to indicate the error.
                IF _scalingReadState = UINT#25 THEN
                    IF PNU_12694 = 16640 AND PNU_12695 = 16643 AND PNU_12696 = 16727 AND PNU_12697 = 16800 THEN
                        AxisType := eAxoDriveAxisType#Rotary;
                        _scalingReadState := UINT#26;
                    ELSIF PNU_12694 = 256 AND PNU_12695 = 259 AND PNU_12696 = 343 AND PNU_12697 = 416 THEN
                        AxisType := eAxoDriveAxisType#Linear;
                        _scalingReadState := UINT#26;
                    ELSE
                        AxisType := eAxoDriveAxisType#Error;
                        Messenger.Activate(ULINT#1801 , eAxoMessageCategory#Error);
                    END_IF;
                END_IF;
                IF _scalingReadState = UINT#26 THEN
                    IF AxisType = eAxoDriveAxisType#Rotary THEN
                        _scalingReadState := UINT#27;
                    ELSIF AxisType = eAxoDriveAxisType#Linear THEN
                        _scalingReadState := UINT#28;
                    END_IF;
                END_IF;
                //Rotary
                IF _scalingReadState = UINT#27 THEN
                    ScalingConstantRequiredPosition := _exp[-1*(TO_INT(PNU_11724) )];               // TODO verify scaling with Automation Suite
                    ScalingConstantActualPosition := LREAL#1.0/ScalingConstantRequiredPosition;     // TODO verify scaling with Automation Suite

                    ScalingConstantRequiredVelocity :=  _exp[-1*(TO_INT(PNU_11725) )];                // TODO verify scaling with Automation Suite
                    ScalingConstantActualVelocity := PNU_12345 * _exp[(TO_INT(PNU_11725) + 3)] / LREAL#1073741824.0;  //  16#4000 0000 ~~ 1073741824    // TODO verify scaling with Automation Suite

                    ScalingConstantRequiredAcceleration := LREAL#16384.0 * _exp[TO_INT(PNU_11726)+3] / PNU_810;  //  16#4000 ~~ 16384
                    ScalingConstantActualAcceleration := LREAL#1.0 / ScalingConstantRequiredAcceleration;

                    ScalingConstantRequiredDeceleration := LREAL#16384.0 * _exp[TO_INT(PNU_11726)+3] / PNU_811; //  16#4000 ~~ 16384
                    ScalingConstantActualDeceleration := LREAL#1.0 / ScalingConstantRequiredDeceleration;

                    ScalingConstantRequiredTorque := 1;
                    ScalingConstantActualTorque := PNU_11122 / 16384; //  16#4000 ~~ 16384

                    ScalingConstantRequiredJerk := _exp[TO_INT(PNU_11727)+3];
                    ScalingConstantActualJerk := LREAL#1.0 / ScalingConstantRequiredJerk;

                    _scalingReadState := UINT#29;
                END_IF;
                //Linear
                IF _scalingReadState = UINT#28 THEN
                    ScalingConstantRequiredPosition := _exp[-1*(TO_INT(PNU_11724) + 3)];
                    ScalingConstantActualPosition := LREAL#1.0/ScalingConstantRequiredPosition;

                    ScalingConstantRequiredVelocity :=  _exp[-1*(TO_INT(PNU_11725) + 3)];
                    ScalingConstantActualVelocity := PNU_12345 * _exp[(TO_INT(PNU_11725) + 6)] / LREAL#1073741824.0;  //  16#4000 0000 ~~ 1073741824

                    ScalingConstantRequiredAcceleration := LREAL#16384.0 * _exp[TO_INT(PNU_11726)] / PNU_810;  //  16#4000 ~~ 16384
                    ScalingConstantActualAcceleration := LREAL#1.0 / ScalingConstantRequiredAcceleration;

                    ScalingConstantRequiredDeceleration := LREAL#16384.0 * _exp[TO_INT(PNU_11726)] / PNU_811; //  16#4000 ~~ 16384
                    ScalingConstantActualDeceleration := LREAL#1.0 / ScalingConstantRequiredDeceleration;

                    ScalingConstantRequiredTorque := 1;
                    ScalingConstantActualTorque := PNU_11122 / 16384; //  16#4000 ~~ 16384

                    ScalingConstantRequiredJerk := _exp[TO_INT(PNU_11727)];
                    ScalingConstantActualJerk := LREAL#1.0 / ScalingConstantRequiredJerk;

                    _scalingReadState := UINT#29;
                END_IF;

                IF _scalingReadState = UINT#29 THEN

                    _ScalingRead := TRUE;
                    _scalingReadState := UINT#0;
                    State := UINT#0;

                    AxoStop_Deceleration := 1000.0;         // mm/s2
                    AxoStop_Jerk := 150000.0;               // mm/s3
                    AxoHalt_Deceleration := 1000.0;         // mm/s2
                    AxoHalt_Jerk := 150000.0;               // mm/s3
                    AxoHome_Position := 0.0;                // mm
                    AxoHome_HommingMode := 1;               // Negative hardware limit switch with zero pulse
                    AxoHome_Velocity := 2.0;                // mm/s
                    AxoHome_Acceleration := 1000.0;         // mm/s2
                    AxoHome_Deceleration := 1000.0;         // mm/s2
                    AxoSetPosition_Position := 0.0;         // mm
                    AxoMoveAbsolute_Position := 0.0;        // mm
                    AxoMoveAbsolute_Velocity := 5.0;        // mm/s
                    AxoMoveAbsolute_Acceleration := 1000.0; // mm/s2
                    AxoMoveAbsolute_Deceleration := 1000.0; // mm/s2
                    AxoMoveAbsolute_Jerk := 150000.0;       // mm/s3
                    AxoMoveRelative_Distance := 5.0;        // mm
                    AxoMoveRelative_Velocity := 5.0;        // mm/s
                    AxoMoveRelative_Acceleration := 1000.0; // mm/s2
                    AxoMoveRelative_Deceleration := 1000.0; // mm/s2
                    AxoMoveRelative_Jerk := 150000.0;       // mm/s3
                    AxoMoveAdditive_Distance := 5.0;        // mm
                    AxoMoveAdditive_Velocity := 5.0;        // mm/s
                    AxoMoveAdditive_Acceleration := 1000.0; // mm/s2
                    AxoMoveAdditive_Deceleration := 1000.0; // mm/s2
                    AxoMoveAdditive_Jerk := 150000.0;       // mm/s3
                    AxoMoveVelocity_Velocity := 5.0;        // mm/s
                    AxoMoveVelocity_Acceleration := 1000.0; // mm/s2
                    AxoMoveVelocity_Deceleration := 1000.0; // mm/s2
                    AxoMoveVelocity_Jerk := 150000.0;       // mm/s3
                    AxoTorqueControl_Torque := 0.0;         // Nm
                    AxoTorqueControl_TorqueRamp := 1.0;     // Nm/s
                    AxoTorqueControl_Velocity := 5.0;       // mm/s
                    AxoTorqueControl_Acceleration := 1000.0;// mm/s2
                    AxoTorqueControl_Deceleration := 1000.0;// mm/s2
                    AxoTorqueControl_Jerk := 150000.0;      // mm/s3
                    AxoJog_Velocity := 2.0;                 // mm/s
                    AxoJog_Acceleration := 500.0;           // mm/s2
                    AxoJog_Deceleration := 500.0;           // mm/s2
                    AxoJog_Jerk := 150000.0;                // mm/s3
                END_IF;
                RETURN;
            END_IF;
            //*************************************************//

            Messenger.ActivateOnCondition(ULINT#300, Enable AND NOT EnablePositive, eAxoMessageCategory#Info);
            Messenger.ActivateOnCondition(ULINT#301, Enable AND NOT EnableNegative, eAxoMessageCategory#Info);

            //************************************************************
            SUPER.Run(THIS,AxisRefExt,Enable,EnablePositive,EnableNegative);
            //************************************************************

            THIS.ActualPosition := TO_LREAL(AxisRefExt.Telegram111_In.XIST_A) * ScalingConstantActualPosition;
            THIS.ActualVelocity := TO_LREAL(AxisRefExt.Telegram111_In.NIST_B) * ScalingConstantActualVelocity;
            THIS.ActualTorque := TO_LREAL(AxisRefExt.Telegram750_In.M_Actual) * ScalingConstantActualTorque;

            IF NOT AxisRefExt.Telegram111_In.ZSW1.operationEnabled THEN
                DriveState := AXOpen.Components.Drives.eAxoDriveState#Disabled;
            ELSIF State>=UINT#20 AND State<UINT#59 OR AxisRefExt.Telegram111_Out.STW1.StartHoming THEN// AxisRef^.Fieldbus_Out.DriveToZeroPoint
                DriveState := AXOpen.Components.Drives.eAxoDriveState#Homing;
            ELSIF State>=UINT#80 AND State<UINT#109 THEN
                DriveState := AXOpen.Components.Drives.eAxoDriveState#DiscreteMotion;
            ELSIF State>=UINT#110 AND State<UINT#129 THEN
                DriveState := AXOpen.Components.Drives.eAxoDriveState#ContinuousMotion;
            // ELSIF _AxisReference^.Data.SynchronizedMotion THEN
            //     DriveState := AXOpen.Components.Drives.eAxoDriveState#SynchronizedMotion;
            ELSIF NOT AxisRefExt.Telegram111_Out.STW1.cancelTraversing AND NOT AxisRefExt.Telegram111_In.ZSW1.driveStopped THEN
                DriveState := AXOpen.Components.Drives.eAxoDriveState#Stopping;
            ELSIF AxisRefExt.Telegram111_In.ZSW1.faultPresent AND AxisRefExt.Telegram111_In.ZSW1.driveStopped THEN
                DriveState := AXOpen.Components.Drives.eAxoDriveState#Errorstop;
            ELSIF AxisRefExt.Telegram111_In.ZSW1.driveStopped THEN
                DriveState := AXOpen.Components.Drives.eAxoDriveState#Standstill;
            END_IF;

        END_METHOD

        ///<summary>
        /// Ensures swapping the hardware input data structure into the AxisRef data structure
        ///</summary>
        METHOD PROTECTED OVERRIDE UpdateInputs : BOOL
            VAR_INPUT
                AxisRef             :   AXOpen.Components.Abstractions.Drives.IAxoAxisReference;
            END_VAR
            VAR
                _AxisReference :  REF_TO AXOpen.Components.Festo.Drives.AxoCmmtAsAxisReference;
                _Telegram111 : ARRAY[0..23] OF BYTE;
                _Telegram750 : ARRAY[0..1] OF WORD;
                returnValue : WORD;
            END_VAR

            _AxisReference ?= AxisRef;

            IF(_AxisReference = NULL) THEN
                Messenger.Activate(     UINT#1410, eAxoMessageCategory#ProgrammingError);
                DriveStatus.Error.Id := UINT#1410;
                RETURN;
            END_IF;

            returnValue := Siemens.Simatic.DistributedIO.ReadData(_AxisReference^.HWIDs.HW_Telegram111 ,_Telegram111);
            IF returnValue > WORD#0 THEN
                Messenger.Activate(     UINT#1411, eAxoMessageCategory#Error);
                DriveStatus.Error.Id := UINT#1411;
                RETURN;
            END_IF;

            // ZSW1
            _AxisReference^.Telegram111_In.ZSW1.followingErrorInTolerance             := _Telegram111[0].%X0; //.8
            _AxisReference^.Telegram111_In.ZSW1.controlRequest                        := _Telegram111[0].%X1; //.9
            _AxisReference^.Telegram111_In.ZSW1.targetPosReached                      := _Telegram111[0].%X2; //.10
            _AxisReference^.Telegram111_In.ZSW1.homePosSet                            := _Telegram111[0].%X3; //.11
            _AxisReference^.Telegram111_In.ZSW1.acknowledgeTraversingBlockActivated   := _Telegram111[0].%X4; //.12
            _AxisReference^.Telegram111_In.ZSW1.driveStopped                          := _Telegram111[0].%X5; //.13
            _AxisReference^.Telegram111_In.ZSW1.axisAccelerates                       := _Telegram111[0].%X6; //.14
            _AxisReference^.Telegram111_In.ZSW1.axisDecelerates                       := _Telegram111[0].%X7; //.15
            _AxisReference^.Telegram111_In.ZSW1.readyForSwitchOn                      := _Telegram111[1].%X0; //.0
            _AxisReference^.Telegram111_In.ZSW1.ready                                 := _Telegram111[1].%X1; //.1
            _AxisReference^.Telegram111_In.ZSW1.operationEnabled                      := _Telegram111[1].%X2; //.2
            _AxisReference^.Telegram111_In.ZSW1.faultPresent                          := _Telegram111[1].%X3; //.3
            _AxisReference^.Telegram111_In.ZSW1.noCoastingActive                      := _Telegram111[1].%X4; //.4
            _AxisReference^.Telegram111_In.ZSW1.noQuickStopActive                     := _Telegram111[1].%X5; //.5
            _AxisReference^.Telegram111_In.ZSW1.switchingOnInhibitedActive            := _Telegram111[1].%X6; //.6
            _AxisReference^.Telegram111_In.ZSW1.warningActive                         := _Telegram111[1].%X7; //.7
            //POS_ZSW1
            _AxisReference^.Telegram111_In.POS_ZSW1.%B1                               := _Telegram111[2];
            _AxisReference^.Telegram111_In.POS_ZSW1.%B0                               := _Telegram111[3];
            // Positioning.Outputs.EPosZSW1 := _AxisReference^.Telegram111_In.POS_ZSW1;
            //POS_ZSW2
            _AxisReference^.Telegram111_In.POS_ZSW2.%B1                               := _Telegram111[4];
            _AxisReference^.Telegram111_In.POS_ZSW2.%B0                               := _Telegram111[5];
            // Positioning.Outputs.EPosZSW2 := _AxisReference^.Telegram111_In.POS_ZSW2;
            // ZSW2
            _AxisReference^.Telegram111_In.ZSW2.deviceSpecificBit8                    := _Telegram111[6].%X0;
            _AxisReference^.Telegram111_In.ZSW2.deviceSpecificBit9                    := _Telegram111[6].%X1;
            _AxisReference^.Telegram111_In.ZSW2.deviceSpecificBit10                   := _Telegram111[6].%X2;
            _AxisReference^.Telegram111_In.ZSW2.deviceSpecificBit11                   := _Telegram111[6].%X3;
            _AxisReference^.Telegram111_In.ZSW2.doSignOfLifeBit0                      := _Telegram111[6].%X4;
            _AxisReference^.Telegram111_In.ZSW2.doSignOfLifeBit1                      := _Telegram111[6].%X5;
            _AxisReference^.Telegram111_In.ZSW2.doSignOfLifeBit2                      := _Telegram111[6].%X6;
            _AxisReference^.Telegram111_In.ZSW2.doSignOfLifeBit3                      := _Telegram111[6].%X7;
            _AxisReference^.Telegram111_In.ZSW2.deviceSpecificBit0                    := _Telegram111[7].%X0;
            _AxisReference^.Telegram111_In.ZSW2.deviceSpecificBit1                    := _Telegram111[7].%X1;
            _AxisReference^.Telegram111_In.ZSW2.deviceSpecificBit2                    := _Telegram111[7].%X2;
            _AxisReference^.Telegram111_In.ZSW2.deviceSpecificBit3                    := _Telegram111[7].%X3;
            _AxisReference^.Telegram111_In.ZSW2.deviceSpecificBit4                    := _Telegram111[7].%X4;
            _AxisReference^.Telegram111_In.ZSW2.deviceSpecificBit5                    := _Telegram111[7].%X5;
            _AxisReference^.Telegram111_In.ZSW2.deviceSpecificBit6                    := _Telegram111[7].%X6;
            _AxisReference^.Telegram111_In.ZSW2.deviceSpecificBit7                    := _Telegram111[7].%X7;
            //MELDW
            _AxisReference^.Telegram111_In.MELDW.%B1                                  := _Telegram111[8];
            _AxisReference^.Telegram111_In.MELDW.%B0                                  := _Telegram111[9];
            //XIST_A
            _AxisReference^.Telegram111_In.XIST_A.%B3                                 := _Telegram111[10];
            _AxisReference^.Telegram111_In.XIST_A.%B2                                 := _Telegram111[11];
            _AxisReference^.Telegram111_In.XIST_A.%B1                                 := _Telegram111[12];
            _AxisReference^.Telegram111_In.XIST_A.%B0                                 := _Telegram111[13];
            //NIST_B
            _AxisReference^.Telegram111_In.NIST_B.%B3                                 := _Telegram111[14];
            _AxisReference^.Telegram111_In.NIST_B.%B2                                 := _Telegram111[15];
            _AxisReference^.Telegram111_In.NIST_B.%B1                                 := _Telegram111[16];
            _AxisReference^.Telegram111_In.NIST_B.%B0                                 := _Telegram111[17];
            //Fault_Code
            _AxisReference^.Telegram111_In.Fault_Code.%B1                             := _Telegram111[18];
            _AxisReference^.Telegram111_In.Fault_Code.%B0                             := _Telegram111[19];
            //Warn_Code
            _AxisReference^.Telegram111_In.Warn_Code.%B1                              := _Telegram111[20];
            _AxisReference^.Telegram111_In.Warn_Code.%B0                              := _Telegram111[21];
            //Reserved
            _AxisReference^.Telegram111_In.Reserved.%B1                               := _Telegram111[22];
            _AxisReference^.Telegram111_In.Reserved.%B0                               := _Telegram111[23];
            //M_Actual
            returnValue := Siemens.Simatic.DistributedIO.ReadData(_AxisReference^.HWIDs.HW_Telegram750,_Telegram750);
            IF returnValue > WORD#0 THEN
                Messenger.Activate(     UINT#1412, eAxoMessageCategory#Error);
                DriveStatus.Error.Id := UINT#1412;
                RETURN;
            END_IF;
            _AxisReference^.Telegram750_In.M_Actual                                   := TO_INT(_Telegram750[0]);
        END_METHOD

        ///<summary>
        /// Ensures swapping the AxisRef data structure into the hardware output data structure
        ///</summary>
        METHOD PROTECTED OVERRIDE UpdateOutputs : BOOL
            VAR_INPUT
                AxisRef             :   AXOpen.Components.Abstractions.Drives.IAxoAxisReference;
            END_VAR
            VAR
                _AxisReference :  REF_TO AXOpen.Components.Festo.Drives.AxoCmmtAsAxisReference;
                tempDWord   :   DWORD;
                _Telegram111 : ARRAY[0..23] OF BYTE;
                _Telegram750 : ARRAY[0..7] OF BYTE;
                returnValue : WORD;
            END_VAR
            _AxisReference ?= AxisRef;

            IF(_AxisReference = NULL) THEN
                Messenger.Activate(     UINT#1420, eAxoMessageCategory#ProgrammingError);
                DriveStatus.Error.Id := UINT#1420;
                RETURN;
            END_IF;

            //STW1
            _Telegram111[1].%X0 := _AxisReference^.Telegram111_Out.STW1.on_;
            _Telegram111[1].%X1 := _AxisReference^.Telegram111_Out.STW1.noCoastStop;
            _Telegram111[1].%X2 := _AxisReference^.Telegram111_Out.STW1.noQuickStop;
            _Telegram111[1].%X3 := _AxisReference^.Telegram111_Out.STW1.enableOperation;
            _Telegram111[1].%X4 := _AxisReference^.Telegram111_Out.STW1.cancelTraversing;
            _Telegram111[1].%X5 := _AxisReference^.Telegram111_Out.STW1.intermediateStop;
            _Telegram111[1].%X6 := _AxisReference^.Telegram111_Out.STW1.activateTraversing;
            _Telegram111[1].%X7 := _AxisReference^.Telegram111_Out.STW1.acknowledgeFault;
            _Telegram111[0].%X0 := _AxisReference^.Telegram111_Out.STW1.jog1;
            _Telegram111[0].%X1 := _AxisReference^.Telegram111_Out.STW1.jog2;
            _Telegram111[0].%X2 := _AxisReference^.Telegram111_Out.STW1.controlByPlc;
            _Telegram111[0].%X3 := _AxisReference^.Telegram111_Out.STW1.StartHoming;
            _Telegram111[0].%X4 := _AxisReference^.Telegram111_Out.STW1.ReleaseBrake;
            _Telegram111[0].%X5 := _AxisReference^.Telegram111_Out.STW1.ExternalBlockChange;
            _Telegram111[0].%X6 := _AxisReference^.Telegram111_Out.STW1.reserved14;
            _Telegram111[0].%X7 := _AxisReference^.Telegram111_Out.STW1.reserved15;
            //POS_STW1
            _Telegram111[3].%X0 := _AxisReference^.Telegram111_Out.POS_STW1.travBlockBit0;
            _Telegram111[3].%X1 := _AxisReference^.Telegram111_Out.POS_STW1.travBlockBit1;
            _Telegram111[3].%X2 := _AxisReference^.Telegram111_Out.POS_STW1.travBlockBit2;
            _Telegram111[3].%X3 := _AxisReference^.Telegram111_Out.POS_STW1.travBlockBit3;
            _Telegram111[3].%X4 := _AxisReference^.Telegram111_Out.POS_STW1.travBlockBit4;
            _Telegram111[3].%X5 := _AxisReference^.Telegram111_Out.POS_STW1.travBlockBit5;
            _Telegram111[3].%X6 := _AxisReference^.Telegram111_Out.POS_STW1.travBlockBit6;
            _Telegram111[3].%X7 := _AxisReference^.Telegram111_Out.POS_STW1.reserved7;
            _Telegram111[2].%X0 := _AxisReference^.Telegram111_Out.POS_STW1.MDI_MOD;
            _Telegram111[2].%X1 := _AxisReference^.Telegram111_Out.POS_STW1.PosModulo;
            _Telegram111[2].%X2 := _AxisReference^.Telegram111_Out.POS_STW1.NegModulo;
            _Telegram111[2].%X3 := _AxisReference^.Telegram111_Out.POS_STW1.reserved11;
            _Telegram111[2].%X4 := _AxisReference^.Telegram111_Out.POS_STW1.reserved12;
            _Telegram111[2].%X5 := _AxisReference^.Telegram111_Out.POS_STW1.reserved13;
            _Telegram111[2].%X6 := _AxisReference^.Telegram111_Out.POS_STW1.SetupMode;
            _Telegram111[2].%X7 := _AxisReference^.Telegram111_Out.POS_STW1.MDI_Activate;
            //POS_STW2
            _Telegram111[5].%X0 := _AxisReference^.Telegram111_Out.POS_STW2.Trackingmode;
            _Telegram111[5].%X1 := _AxisReference^.Telegram111_Out.POS_STW2.SetReferencePoint;
            _Telegram111[5].%X2 := _AxisReference^.Telegram111_Out.POS_STW2.reserved2;
            _Telegram111[5].%X3 := _AxisReference^.Telegram111_Out.POS_STW2.reserved3;
            _Telegram111[5].%X4 := _AxisReference^.Telegram111_Out.POS_STW2.reserved4;
            _Telegram111[5].%X5 := _AxisReference^.Telegram111_Out.POS_STW2.jog_inc;
            _Telegram111[5].%X6 := _AxisReference^.Telegram111_Out.POS_STW2.reserved6;
            _Telegram111[5].%X7 := _AxisReference^.Telegram111_Out.POS_STW2.reserved7;
            _Telegram111[4].%X0 := _AxisReference^.Telegram111_Out.POS_STW2.FlyingRef;
            _Telegram111[4].%X1 := _AxisReference^.Telegram111_Out.POS_STW2.reserved9;
            _Telegram111[4].%X2 := _AxisReference^.Telegram111_Out.POS_STW2.SelectProbe;
            _Telegram111[4].%X3 := _AxisReference^.Telegram111_Out.POS_STW2.ProbeEdgeEval;
            _Telegram111[4].%X4 := _AxisReference^.Telegram111_Out.POS_STW2.reserved12;
            _Telegram111[4].%X5 := _AxisReference^.Telegram111_Out.POS_STW2.reserved13;
            _Telegram111[4].%X6 := _AxisReference^.Telegram111_Out.POS_STW2.SW_Limit;
            _Telegram111[4].%X7 := _AxisReference^.Telegram111_Out.POS_STW2.HW_Limit;
            //STW2
            _Telegram111[7].%X0 := _AxisReference^.Telegram111_Out.STW2.reserved0;
            _Telegram111[7].%X1 := _AxisReference^.Telegram111_Out.STW2.reserved1;
            _Telegram111[7].%X2 := _AxisReference^.Telegram111_Out.STW2.reserved2;
            _Telegram111[7].%X3 := _AxisReference^.Telegram111_Out.STW2.reserved3;
            _Telegram111[7].%X4 := _AxisReference^.Telegram111_Out.STW2.reserved4;
            _Telegram111[7].%X5 := _AxisReference^.Telegram111_Out.STW2.reserved5;
            _Telegram111[7].%X6 := _AxisReference^.Telegram111_Out.STW2.reserved6;
            _Telegram111[7].%X7 := _AxisReference^.Telegram111_Out.STW2.reserved7;
            _Telegram111[6].%X0 := _AxisReference^.Telegram111_Out.STW2.TravelToFixStop;
            _Telegram111[6].%X1 := _AxisReference^.Telegram111_Out.STW2.reserved9;
            _Telegram111[6].%X2 := _AxisReference^.Telegram111_Out.STW2.reserved10;
            _Telegram111[6].%X3 := _AxisReference^.Telegram111_Out.STW2.reserved11;
            _Telegram111[6].%X4 := _AxisReference^.Telegram111_Out.STW2.signOfLifeBit0;
            _Telegram111[6].%X5 := _AxisReference^.Telegram111_Out.STW2.signOfLifeBit1;
            _Telegram111[6].%X6 := _AxisReference^.Telegram111_Out.STW2.signOfLifeBit2;
            _Telegram111[6].%X7 := _AxisReference^.Telegram111_Out.STW2.signOfLifeBit3;
            //Override
            _Telegram111[9] := _AxisReference^.Telegram111_Out.Override_.%B0;
            _Telegram111[8] := _AxisReference^.Telegram111_Out.Override_.%B1;
            //TargetPos
            tempDWord := TO_DWORD(_AxisReference^.Telegram111_Out.MDI_TARPOS);
            _Telegram111[13] := tempDWord.%B0;
            _Telegram111[12] := tempDWord.%B1;
            _Telegram111[11] := tempDWord.%B2;
            _Telegram111[10] := tempDWord.%B3;
            //TargetVelocity
            tempDWord := TO_DWORD(_AxisReference^.Telegram111_Out.MDI_VELOCITY);
            _Telegram111[17] := tempDWord.%B0;
            _Telegram111[16] := tempDWord.%B1;
            _Telegram111[15] := tempDWord.%B2;
            _Telegram111[14] := tempDWord.%B3;
            // ACC, DEC
            _Telegram111[19] := _AxisReference^.Telegram111_Out.MDI_ACC.%B0;
            _Telegram111[18] := _AxisReference^.Telegram111_Out.MDI_ACC.%B1;
            _Telegram111[21] := _AxisReference^.Telegram111_Out.MDI_DEC.%B0;
            _Telegram111[20] := _AxisReference^.Telegram111_Out.MDI_DEC.%B1;
            _Telegram111[23] := _AxisReference^.Telegram111_Out.reserved11.%B0;
            _Telegram111[22] := _AxisReference^.Telegram111_Out.reserved11.%B1;

            returnValue := Siemens.Simatic.DistributedIO.WriteData(_AxisReference^.HWIDs.HW_Telegram111,_Telegram111);
            IF returnValue > WORD#0 THEN
                Messenger.Activate(     UINT#1421, eAxoMessageCategory#Error);
                DriveStatus.Error.Id := UINT#1421;
                RETURN;
            END_IF;
            // M_ADD1, M_LIMIT_POS, M_LIMIT_NEG
            _Telegram750[1] := _AxisReference^.Telegram750_Out.M_ADD1.%B0;
            _Telegram750[0] := _AxisReference^.Telegram750_Out.M_ADD1.%B1;
            _Telegram750[3] := _AxisReference^.Telegram750_Out.M_LIMIT_POS.%B0;
            _Telegram750[2] := _AxisReference^.Telegram750_Out.M_LIMIT_POS.%B1;
            _Telegram750[5] := _AxisReference^.Telegram750_Out.M_LIMIT_NEG.%B0;
            _Telegram750[4] := _AxisReference^.Telegram750_Out.M_LIMIT_NEG.%B1;
            _Telegram750[7] := _AxisReference^.Telegram750_Out.Reserved.%B0;
            _Telegram750[6] := _AxisReference^.Telegram750_Out.Reserved.%B1;

            returnValue := Siemens.Simatic.DistributedIO.WriteData(_AxisReference^.HWIDs.HW_Telegram750,_Telegram750);
            IF returnValue > WORD#0 THEN
                Messenger.Activate(     UINT#1422, eAxoMessageCategory#Error);
                DriveStatus.Error.Id := UINT#1422;
                RETURN;
            END_IF;

        END_METHOD

        ///<summary>
        /// This method controls the power stage (On or Off).
        ///</summary>
        VAR INTERNAL
            MC_PowerEnable_PV					:	BOOL := FALSE;		//Enable - previous value
            MC_PowerCycle					    :	ULINT   := ULINT#0;
        END_VAR
        METHOD PUBLIC OVERRIDE MC_Power
            VAR_INPUT
                AxisRef         :   AXOpen.Components.Abstractions.Drives.IAxoAxisReference;
                Enable          :   BOOL;                       //  As long as ‘Enable’ is true, power is being enabled.
            END_VAR
            VAR_OUTPUT
                Status          :   BOOL;                       //  Effective state of the power stage
                Valid           :   BOOL;                       //  If true, a valid set of outputs is available at the method
                Error           :   BOOL;                       //  Signals that an error has occurred within the method
                ErrorID         :   DINT;                       //  Error identification
            END_VAR
            VAR
                _AxisReference :  REF_TO AXOpen.Components.Festo.Drives.AxoCmmtAsAxisReference;
                Dummy : BOOL;
            END_VAR

            _AxisReference ?= AxisRef;

            IF(_AxisReference = NULL) THEN
                Messenger.Activate(     UINT#1430, eAxoMessageCategory#ProgrammingError);
                DriveStatus.Error.Id := UINT#1430;
                RETURN;
            END_IF;

            IF Enable THEN
                MC_PowerCycle := MC_PowerCycle + ULINT#1;
                THIS.UpdateInputs(AxisRef);

                IF NOT MC_PowerEnable_PV THEN
                    _AxisReference^.Telegram750_Out.M_LIMIT_POS := 16384;
                    _AxisReference^.Telegram750_Out.M_LIMIT_NEG := -16384;
                    _AxisReference^.Telegram111_Out.MDI_ACC := TO_UINT(16384.0 * _AxisReference^.Data.OverrideAccelerationFactor);
                    _AxisReference^.Telegram111_Out.MDI_DEC := TO_UINT(16384.0 * _AxisReference^.Data.OverrideAccelerationFactor);
                    _AxisReference^.Telegram111_Out.Override_ := TO_WORD(TO_INT(16384.0 )); // * _AxisReference^.Data.OverrideVelocityFactor));
                    _AxisReference^.Telegram111_Out.MDI_VELOCITY := DINT#1;
                END_IF;
                _AxisReference^.Telegram111_Out.STW1.on_ := TRUE;
                _AxisReference^.Telegram111_Out.STW1.activateTraversing := FALSE;
                _AxisReference^.Telegram111_Out.STW1.acknowledgeFault := FALSE;
                // _AxisReference^.Telegram111_Out.MDI_VELOCITY := DINT#1;
                // _AxisReference^.Telegram111_Out.POS_STW2.SW_Limit := TRUE;
                _AxisReference^.Telegram111_Out.POS_STW2.HW_Limit := TRUE;
                _AxisReference^.Telegram111_Out.STW1.noCoastStop := TRUE;
                _AxisReference^.Telegram111_Out.STW1.noQuickStop := TRUE;
                _AxisReference^.Telegram111_Out.STW1.enableOperation := TRUE;
                _AxisReference^.Telegram111_Out.STW1.cancelTraversing := TRUE;
                _AxisReference^.Telegram111_Out.STW1.intermediateStop := TRUE;
                _AxisReference^.Telegram111_Out.STW1.controlByPlc := TRUE;
                IF _AxisReference^.Telegram111_In.ZSW1.operationEnabled THEN
                    MC_PowerCycle := ULINT#0;
                    Status	:= TRUE;						(* Status OK*)
                    Valid := TRUE;
                ELSIF _AxisReference^.Telegram111_In.ZSW1.faultPresent = TRUE THEN
                    Error		:= TRUE; 						(*	Set the ERROR-Output *)
                    Valid := TRUE;
                    ErrorID := TO_DINT(_AxisReference^.Telegram111_In.Fault_Code);
                END_IF;
                IF MC_PowerCycle >= ULINT#2000 THEN
                    MC_PowerCycle := ULINT#0;
                    _AxisReference^.Telegram111_Out.STW1.on_  := FALSE;
                    _AxisReference^.Telegram111_Out.STW1.StartHoming := FALSE;
                    _AxisReference^.Telegram111_Out.POS_STW1.MDI_MOD := FALSE;
                    _AxisReference^.Telegram111_Out.POS_STW1.PosModulo := FALSE;
                    _AxisReference^.Telegram111_Out.POS_STW1.NegModulo := FALSE;
                    _AxisReference^.Telegram111_Out.POS_STW1.SetupMode := FALSE;
                    _AxisReference^.Telegram111_Out.POS_STW1.MDI_Activate := FALSE;
                    _AxisReference^.Telegram111_Out.POS_STW2.Trackingmode := FALSE;
                    _AxisReference^.Telegram111_Out.POS_STW2.jog_inc := FALSE;
                    _AxisReference^.Telegram111_Out.POS_STW1.travBlockBit0 := FALSE;
                    _AxisReference^.Telegram111_Out.POS_STW1.travBlockBit1 := FALSE;
                    _AxisReference^.Telegram111_Out.POS_STW1.travBlockBit2 := FALSE;
                    _AxisReference^.Telegram111_Out.POS_STW1.travBlockBit3 := FALSE;
                    _AxisReference^.Telegram111_Out.POS_STW1.travBlockBit4 := FALSE;
                    _AxisReference^.Telegram111_Out.POS_STW1.travBlockBit5 := FALSE;
                    _AxisReference^.Telegram111_Out.POS_STW1.travBlockBit6 := FALSE;
                    _AxisReference^.Telegram111_Out.STW2.TravelToFixStop := FALSE;
                    _AxisReference^.Telegram111_Out.STW1.acknowledgeFault := TRUE;
                END_IF;
                THIS.UpdateOutputs(AxisRef);
            END_IF;

            IF NOT Enable AND MC_PowerEnable_PV  THEN
                THIS.UpdateInputs(AxisRef);
                MC_PowerCycle := ULINT#0;
                _AxisReference^.Telegram111_Out.STW1.on_  := FALSE;
                THIS.UpdateOutputs(AxisRef);
            END_IF;

            MC_PowerEnable_PV := Enable;
        END_METHOD

        ///<summary>
        /// This method commands the axis to perform the «search home» sequence. The details of this sequence are
        /// manufacturer dependent and can be set by the axis’ parameters. The ‘Position’ input is used to set the absolute
        /// position when reference signal is detected. This method completes at ‘Standstill’ if it was started in ‘Standstill’.
        ///</summary>
        VAR INTERNAL
            MC_HomeExecute_PV					: 	BOOL;				//Execute - previous value
            MC_HomeErrorID					    : 	DINT;
            MC_HomeCycle					    : 	ULINT;
        END_VAR
        METHOD PUBLIC OVERRIDE MC_Home
            VAR_INPUT
                AxisRef         :   AXOpen.Components.Abstractions.Drives.IAxoAxisReference;
                Execute         :   BOOL;                       //  Start the motion at rising edge
                Position        :   LREAL;                      //  Absolute position when the reference signal is detected
                HommingMode     :   INT;                        //  Required homming mode
                Velocity        :   LREAL;                      //  Value of the maximum ‘Velocity’ (not necessarily reached) [u/s].
                Acceleration    :   LREAL;                      //  Value of the ‘Acceleration’ (always positive) (increasing energy of the motor) [u/s2]
                Deceleration    :   LREAL;                      //  Value of the ‘Deceleration’ (always positive) (decreasing energy of the motor) [u/s2]
            END_VAR
            VAR_OUTPUT
                Done            :   BOOL;                       // Reference known and set sucessfully
                Busy            :   BOOL;                       // The method is not finished and new output values are to be expected
                Active          :   BOOL;                       // Indicates that the method has control on the axis
                CommandAborted  :   BOOL;                       // ‘Command’ is aborted by another command
                Error           :   BOOL;                       // Signals that an error has occurred within the method
                ErrorID         :   DINT;                       // Error identification
             END_VAR
             VAR
                _AxisReference :  REF_TO AXOpen.Components.Festo.Drives.AxoCmmtAsAxisReference;
                HommingModeInvalid : BOOL;
            END_VAR

            _AxisReference ?= AxisRef;

            IF(_AxisReference = NULL) THEN
                Messenger.Activate(     UINT#1440, eAxoMessageCategory#ProgrammingError);
                DriveStatus.Error.Id := UINT#1440;
                RETURN;
            END_IF;

            HommingModeInvalid := TRUE;
            IF HommingMode = -27 OR  HommingMode = -23 OR HommingMode = -18 OR  HommingMode = -17 OR  HommingMode = -2 OR  HommingMode = -1 OR HommingMode = 1 OR HommingMode = 2 THEN
                HommingModeInvalid := FALSE;
            ELSIF HommingMode = 7 OR  HommingMode = 11 OR HommingMode = 17 OR  HommingMode = 18 OR  HommingMode = 23 OR  HommingMode = 27 OR HommingMode = 33 OR HommingMode = 34 OR HommingMode = 37 THEN
                HommingModeInvalid := FALSE;
            END_IF;

            Messenger.ActivateOnCondition(ULINT#1441, Execute AND Acceleration <= 0, eAxoMessageCategory#ProgrammingError);
            Messenger.ActivateOnCondition(ULINT#1442, Execute AND Deceleration <= 0, eAxoMessageCategory#ProgrammingError);
            Messenger.ActivateOnCondition(ULINT#1443, Execute AND HommingModeInvalid, eAxoMessageCategory#ProgrammingError);

            IF THIS.AxoHome_Task.StartTriggered() THEN
                _AxisReference^.Status.CurrentMotionTaskId := AXOpen.Components.Drives.eAxoMotionTaskId#Axo_Home;
            END_IF;

            IF Execute AND NOT MC_HomeExecute_PV AND State = UINT#0 THEN
                _AxisReference^.Data.Cycle := _AxisReference^.Data.Cycle + ULINT#2;
                MC_HomeCycle := _AxisReference^.Data.Cycle ;
            END_IF;

            IF Execute THEN
                THIS.UpdateInputs(AxisRef);
                IF State = UINT#0 THEN
                    Busy := TRUE;
                    Active := TRUE;
                    MC_HomeErrorID :=  DINT#0;
                    _AxisReference^.Telegram111_Out.STW1.StartHoming := FALSE;
                    _AxisReference^.Telegram111_Out.POS_STW1.MDI_MOD := FALSE;
                    _AxisReference^.Telegram111_Out.POS_STW1.PosModulo := FALSE;
                    _AxisReference^.Telegram111_Out.POS_STW1.NegModulo := FALSE;
                    _AxisReference^.Telegram111_Out.POS_STW1.SetupMode := FALSE;
                    _AxisReference^.Telegram111_Out.POS_STW1.MDI_Activate := FALSE;
                    _AxisReference^.Telegram111_Out.POS_STW2.Trackingmode := FALSE;
                    _AxisReference^.Telegram111_Out.POS_STW2.jog_inc := FALSE;
                    _AxisReference^.Telegram111_Out.POS_STW1.travBlockBit0 := FALSE;
                    _AxisReference^.Telegram111_Out.POS_STW1.travBlockBit1 := FALSE;
                    _AxisReference^.Telegram111_Out.POS_STW1.travBlockBit2 := FALSE;
                    _AxisReference^.Telegram111_Out.POS_STW1.travBlockBit3 := FALSE;
                    _AxisReference^.Telegram111_Out.POS_STW1.travBlockBit4 := FALSE;
                    _AxisReference^.Telegram111_Out.POS_STW1.travBlockBit5 := FALSE;
                    _AxisReference^.Telegram111_Out.POS_STW1.travBlockBit6 := FALSE;
                    _AxisReference^.Telegram111_Out.STW2.TravelToFixStop := FALSE;
                    Parametrization.Inputs.Enable := FALSE;
                    State := UINT#20;
                END_IF;

                IF State = UINT#20 THEN
                    IF Acceleration <= 0 OR Deceleration <= 0 OR HommingModeInvalid THEN
                        State := UINT#59;
                    ELSE
                        State := UINT#21;
                    END_IF;
                END_IF;
                //Write  PNU 11206 Acceleration
                IF State = UINT#21 THEN
                    Busy := TRUE;
                    Active := TRUE;
                    Parametrization.Inputs.Enable := TRUE;
                    Parametrization.Inputs.ReadWrite   := TRUE;
                    Parametrization.Inputs.ParameterNo := 11206; //Acc
                    Parametrization.Inputs.Subindex    := 0;
                    Parametrization.Inputs.AxisNo  := BYTE#1;
                    Parametrization.Inputs.HardwareId  := _AxisReference^.HWIDs.HW_ModuleAccessPoint;
                    Parametrization.Inputs.ValueWriteREAL := TO_REAL(Acceleration * ScalingConstantRequiredAcceleration * 0.001);
                    IF Parametrization.Outputs.Done AND NOT Parametrization.Outputs.Error THEN
                        State := UINT#22;
                    END_IF;
                    IF Parametrization.Outputs.Error THEN
                        Messenger.Activate( UINT#1444, eAxoMessageCategory#Error);
                        MC_HomeErrorID :=   DINT#1444;
                        State := UINT#59;
                    END_IF;
                END_IF;
                IF State = UINT#22 THEN
                    Busy := TRUE;
                    Active := TRUE;
                    Parametrization.Inputs.Enable := FALSE;
                    IF  NOT Parametrization.Outputs.Done THEN
                        State := UINT#23;
                    END_IF;
                END_IF;
                //Write  PNU 11209 Acceleration
                IF State = UINT#23 THEN
                    Busy := TRUE;
                    Active := TRUE;
                    Parametrization.Inputs.Enable := TRUE;
                    Parametrization.Inputs.ReadWrite   := TRUE;
                    Parametrization.Inputs.ParameterNo := 11209;//Acc
                    Parametrization.Inputs.Subindex    := 0;
                    Parametrization.Inputs.AxisNo  := BYTE#1;
                    Parametrization.Inputs.HardwareId  := _AxisReference^.HWIDs.HW_ModuleAccessPoint;
                    Parametrization.Inputs.ValueWriteREAL := TO_REAL(Acceleration * ScalingConstantRequiredAcceleration * 0.001);
                    IF Parametrization.Outputs.Done AND NOT Parametrization.Outputs.Error THEN
                        State := UINT#24;
                    END_IF;
                    IF Parametrization.Outputs.Error THEN
                        Messenger.Activate( UINT#1445, eAxoMessageCategory#Error);
                        MC_HomeErrorID :=   DINT#1445;
                        State := UINT#59;
                    END_IF;
                END_IF;
                IF State = UINT#24 THEN
                    Busy := TRUE;
                    Active := TRUE;
                    Parametrization.Inputs.Enable := FALSE;
                    IF  NOT Parametrization.Outputs.Done THEN
                        State := UINT#25;
                    END_IF;
                END_IF;
                //Write  PNU 11728 Acceleration
                IF State = UINT#25 THEN
                    Busy := TRUE;
                    Active := TRUE;
                    Parametrization.Inputs.Enable := TRUE;
                    Parametrization.Inputs.ReadWrite   := TRUE;
                    Parametrization.Inputs.ParameterNo := 11728;//Acc
                    Parametrization.Inputs.Subindex    := 0;
                    Parametrization.Inputs.AxisNo  := BYTE#1;
                    Parametrization.Inputs.HardwareId  := _AxisReference^.HWIDs.HW_ModuleAccessPoint;
                    Parametrization.Inputs.ValueWriteREAL := TO_REAL(Acceleration * ScalingConstantRequiredAcceleration * 0.001);
                    IF Parametrization.Outputs.Done AND NOT Parametrization.Outputs.Error THEN
                        State := UINT#26;
                    END_IF;
                    IF Parametrization.Outputs.Error THEN
                        Messenger.Activate( UINT#1446, eAxoMessageCategory#Error);
                        MC_HomeErrorID :=   DINT#1446;
                        State := UINT#59;
                    END_IF;
                END_IF;
                IF State = UINT#26 THEN
                    Busy := TRUE;
                    Active := TRUE;
                    Parametrization.Inputs.Enable := FALSE;
                    IF  NOT Parametrization.Outputs.Done THEN
                        State := UINT#27;
                    END_IF;
                END_IF;
                //Write  PNU 11205 Velocity
                IF State = UINT#27 THEN
                    Busy := TRUE;
                    Active := TRUE;
                    Parametrization.Inputs.Enable := TRUE;
                    Parametrization.Inputs.ReadWrite   := TRUE;
                    Parametrization.Inputs.ParameterNo := 11205; //Vel
                    Parametrization.Inputs.Subindex    := 0;
                    Parametrization.Inputs.AxisNo  := BYTE#1;
                    Parametrization.Inputs.HardwareId  := _AxisReference^.HWIDs.HW_ModuleAccessPoint;
                    Parametrization.Inputs.ValueWriteREAL := TO_REAL(Velocity * ScalingConstantRequiredVelocity * 0.001);
                    IF Parametrization.Outputs.Done AND NOT Parametrization.Outputs.Error THEN
                        State := UINT#28;
                    END_IF;
                    IF Parametrization.Outputs.Error THEN
                        Messenger.Activate( UINT#1447, eAxoMessageCategory#Error);
                        MC_HomeErrorID :=   DINT#1447;
                        State := UINT#59;
                    END_IF;
                END_IF;
                IF State = UINT#28 THEN
                    Busy := TRUE;
                    Active := TRUE;
                    Parametrization.Inputs.Enable := FALSE;
                    IF  NOT Parametrization.Outputs.Done THEN
                        State := UINT#29;
                    END_IF;
                END_IF;
                //Write  PNU 11208 Velocity
                IF State = UINT#29 THEN
                    Busy := TRUE;
                    Active := TRUE;
                    Parametrization.Inputs.Enable := TRUE;
                    Parametrization.Inputs.ReadWrite   := TRUE;
                    Parametrization.Inputs.ParameterNo := 11208;//Vel
                    Parametrization.Inputs.Subindex    := 0;
                    Parametrization.Inputs.AxisNo  := BYTE#1;
                    Parametrization.Inputs.HardwareId  := _AxisReference^.HWIDs.HW_ModuleAccessPoint;
                    Parametrization.Inputs.ValueWriteREAL := TO_REAL(Velocity* ScalingConstantRequiredVelocity * 0.001)*REAL#0.5;
                    IF Parametrization.Outputs.Done AND NOT Parametrization.Outputs.Error THEN
                        State := UINT#30;
                    END_IF;
                    IF Parametrization.Outputs.Error THEN
                        Messenger.Activate( UINT#1448, eAxoMessageCategory#Error);
                        MC_HomeErrorID :=   DINT#1448;
                        State := UINT#59;
                    END_IF;
                END_IF;
                IF State = UINT#30 THEN
                    Busy := TRUE;
                    Active := TRUE;
                    Parametrization.Inputs.Enable := FALSE;
                    IF  NOT Parametrization.Outputs.Done THEN
                        State := UINT#31;
                    END_IF;
                END_IF;
                //Write  PNU 11211 Velocity
                IF State = UINT#31 THEN
                    Busy := TRUE;
                    Active := TRUE;
                    Parametrization.Inputs.Enable := TRUE;
                    Parametrization.Inputs.ReadWrite   := TRUE;
                    Parametrization.Inputs.ParameterNo := 11211;//Vel
                    Parametrization.Inputs.Subindex    := 0;
                    Parametrization.Inputs.AxisNo  := BYTE#1;
                    Parametrization.Inputs.HardwareId  := _AxisReference^.HWIDs.HW_ModuleAccessPoint;
                    Parametrization.Inputs.ValueWriteREAL := TO_REAL(Velocity * ScalingConstantRequiredVelocity * 0.001)*REAL#5.0;
                    IF Parametrization.Outputs.Done AND NOT Parametrization.Outputs.Error THEN
                        State := UINT#32;
                    END_IF;
                    IF Parametrization.Outputs.Error THEN
                        Messenger.Activate( UINT#1449, eAxoMessageCategory#Error);
                        MC_HomeErrorID :=   DINT#1449;
                        State := UINT#59;
                    END_IF;
                END_IF;
                IF State = UINT#32 THEN
                    Busy := TRUE;
                    Active := TRUE;
                    Parametrization.Inputs.Enable := FALSE;
                    IF  NOT Parametrization.Outputs.Done THEN
                        State := UINT#33;
                    END_IF;
                END_IF;
                //Read  PNU 11735 Homing mode
                IF State = UINT#33 THEN
                    Busy := TRUE;
                    Active := TRUE;
                    Parametrization.Inputs.Enable := TRUE;
                    Parametrization.Inputs.ReadWrite   := FALSE;
                    Parametrization.Inputs.ParameterNo := 11735;//mode
                    Parametrization.Inputs.Subindex    := 0;
                    Parametrization.Inputs.AxisNo  := BYTE#1;
                    Parametrization.Inputs.HardwareId  := _AxisReference^.HWIDs.HW_ModuleAccessPoint;
                    IF Parametrization.Outputs.Done AND NOT Parametrization.Outputs.Error THEN
                        PNU_11735 := Parametrization.Outputs.ValueReadLINT;
                        State := UINT#34;
                    END_IF;
                    IF Parametrization.Outputs.Error THEN
                        Messenger.Activate( UINT#1450, eAxoMessageCategory#Error);
                        MC_HomeErrorID :=   DINT#1450;
                        State := UINT#59;
                    END_IF;
                END_IF;
                IF State = UINT#34 THEN
                    Busy := TRUE;
                    Active := TRUE;
                    Parametrization.Inputs.Enable := FALSE;
                    IF  NOT Parametrization.Outputs.Done THEN
                        State := UINT#35;
                    END_IF;
                END_IF;
                //Write  PNU 11735 Homing mode
                IF State = UINT#35 THEN
                    Busy := TRUE;
                    Active := TRUE;
                    Parametrization.Inputs.Enable := TRUE;
                    Parametrization.Inputs.ReadWrite   := TRUE;
                    Parametrization.Inputs.ParameterNo := 11735;//mode
                    Parametrization.Inputs.Subindex    := 0;
                    Parametrization.Inputs.AxisNo  := BYTE#1;
                    Parametrization.Inputs.HardwareId  := _AxisReference^.HWIDs.HW_ModuleAccessPoint;
                    Parametrization.Inputs.ValueWriteLINT := TO_LINT(HommingMode);
                    IF Parametrization.Outputs.Done AND NOT Parametrization.Outputs.Error THEN
                        State := UINT#36;
                    END_IF;
                    IF Parametrization.Outputs.Error THEN
                        Messenger.Activate( UINT#1451, eAxoMessageCategory#Error);
                        MC_HomeErrorID :=   DINT#1451;
                        State := UINT#59;
                    END_IF;
                END_IF;
                IF State = UINT#36 THEN
                    Busy := TRUE;
                    Active := TRUE;
                    Parametrization.Inputs.Enable := FALSE;
                    IF  NOT Parametrization.Outputs.Done THEN
                        State := UINT#37;
                    END_IF;
                END_IF;
                //Write  PNU 12681 deactivate save zero offset
                IF State = UINT#37 THEN
                    Busy := TRUE;
                    Active := TRUE;
                    Parametrization.Inputs.Enable := TRUE;
                    Parametrization.Inputs.ReadWrite   := TRUE;
                    Parametrization.Inputs.ParameterNo := 12681;//deactivate save zero offset
                    Parametrization.Inputs.Subindex    := 0;
                    Parametrization.Inputs.AxisNo  := BYTE#1;
                    Parametrization.Inputs.HardwareId  := _AxisReference^.HWIDs.HW_ModuleAccessPoint;
                    Parametrization.Inputs.ValueWriteBOOL := FALSE;
                    IF Parametrization.Outputs.Done AND NOT Parametrization.Outputs.Error THEN
                        State := UINT#38;
                    END_IF;
                    IF Parametrization.Outputs.Error THEN
                        Messenger.Activate( UINT#1452, eAxoMessageCategory#Error);
                        MC_HomeErrorID :=   DINT#1452;
                        State := UINT#59;
                    END_IF;
                END_IF;
                IF State = UINT#38 THEN
                    Busy := TRUE;
                    Active := TRUE;
                    Parametrization.Inputs.Enable := FALSE;
                    IF  NOT Parametrization.Outputs.Done THEN
                        State := UINT#39;
                    END_IF;
                END_IF;
                //Homing started
                IF State = UINT#39 THEN
                    Busy := TRUE;
                    Active := TRUE;
                    _AxisReference^.Telegram111_Out.STW1.StartHoming := TRUE;
                    IF  NOT _AxisReference^.Telegram111_In.ZSW1.targetPosReached AND NOT _AxisReference^.Telegram111_In.ZSW1.homePosSet THEN
                        State := UINT#40;
                    END_IF;
                END_IF;
                IF State = UINT#40 THEN
                    Busy := TRUE;
                    Active := TRUE;
                    IF _AxisReference^.Telegram111_In.ZSW1.targetPosReached AND _AxisReference^.Telegram111_In.ZSW1.homePosSet THEN
                        _AxisReference^.Telegram111_Out.STW1.StartHoming := FALSE;
                        IF Position = 0 THEN
                            State := UINT#57;
                        ELSE
                            State := UINT#41;
                        END_IF;
                    END_IF;
                END_IF;
                //Read PNU 11203 Move to axis zero after homming
                IF State = UINT#41 THEN
                    Busy := TRUE;
                    Active := TRUE;
                    Parametrization.Inputs.Enable := TRUE;
                    Parametrization.Inputs.ReadWrite   := FALSE;
                    Parametrization.Inputs.ParameterNo := 11203;//Move to axis zero after homming
                    Parametrization.Inputs.Subindex    := 0;
                    Parametrization.Inputs.AxisNo  := BYTE#1;
                    Parametrization.Inputs.HardwareId  := _AxisReference^.HWIDs.HW_ModuleAccessPoint;
                    IF Parametrization.Outputs.Done AND NOT Parametrization.Outputs.Error THEN
                        PNU_11203 := Parametrization.Outputs.ValueReadBool;
                        State := UINT#42;
                    END_IF;
                    IF Parametrization.Outputs.Error THEN
                        Messenger.Activate( UINT#1453, eAxoMessageCategory#Error);
                        MC_HomeErrorID :=   DINT#1453;
                        State := UINT#59;
                    END_IF;
                END_IF;
                IF State = UINT#42 THEN
                    Busy := TRUE;
                    Active := TRUE;
                    Parametrization.Inputs.Enable := FALSE;
                    IF  NOT Parametrization.Outputs.Done THEN
                        State := UINT#43;
                    END_IF;
                END_IF;
                //Read PNU 11734 Axis zero point offset
                IF State = UINT#43 THEN
                    Busy := TRUE;
                    Active := TRUE;
                    Parametrization.Inputs.Enable := TRUE;
                    Parametrization.Inputs.ReadWrite   := FALSE;
                    Parametrization.Inputs.ParameterNo := 11734;//Move to axis zero after homming
                    Parametrization.Inputs.Subindex    := 0;
                    Parametrization.Inputs.AxisNo  := BYTE#1;
                    Parametrization.Inputs.HardwareId  := _AxisReference^.HWIDs.HW_ModuleAccessPoint;
                    IF Parametrization.Outputs.Done AND NOT Parametrization.Outputs.Error THEN
                        PNU_11734 := Parametrization.Outputs.ValueReadLINT;
                        State := UINT#44;
                    END_IF;
                    IF Parametrization.Outputs.Error THEN
                        Messenger.Activate( UINT#1454, eAxoMessageCategory#Error);
                        MC_HomeErrorID :=   DINT#1454;
                        State := UINT#59;
                    END_IF;
                END_IF;
                IF State = UINT#44 THEN
                    Busy := TRUE;
                    Active := TRUE;
                    Parametrization.Inputs.Enable := FALSE;
                    IF  NOT Parametrization.Outputs.Done THEN
                        State := UINT#45;
                    END_IF;
                END_IF;
                //Write PNU 11203 deactivate Move to axis zero after homming
                IF State = UINT#45 THEN
                    Busy := TRUE;
                    Active := TRUE;
                    Parametrization.Inputs.Enable := TRUE;
                    Parametrization.Inputs.ReadWrite   := TRUE;
                    Parametrization.Inputs.ParameterNo := 11203;//Move to axis zero after homming
                    Parametrization.Inputs.Subindex    := 0;
                    Parametrization.Inputs.AxisNo  := BYTE#1;
                    Parametrization.Inputs.HardwareId  := _AxisReference^.HWIDs.HW_ModuleAccessPoint;
                    Parametrization.Inputs.ValueWriteBOOL := FALSE;
                    IF Parametrization.Outputs.Done AND NOT Parametrization.Outputs.Error THEN
                        State := UINT#46;
                    END_IF;
                    IF Parametrization.Outputs.Error THEN
                        Messenger.Activate( UINT#1455, eAxoMessageCategory#Error);
                        MC_HomeErrorID :=   DINT#1455;
                        State := UINT#59;
                    END_IF;
                END_IF;
                IF State = UINT#46 THEN
                    Busy := TRUE;
                    Active := TRUE;
                    Parametrization.Inputs.Enable := FALSE;
                    IF  NOT Parametrization.Outputs.Done THEN
                        State := UINT#47;
                    END_IF;
                END_IF;
                //Write PNU 11734 Axis zero point offset
                IF State = UINT#47 THEN
                    Busy := TRUE;
                    Active := TRUE;
                    Parametrization.Inputs.Enable := TRUE;
                    Parametrization.Inputs.ReadWrite   := TRUE;
                    Parametrization.Inputs.ParameterNo := 11734;//Move to axis zero after homming
                    Parametrization.Inputs.Subindex    := 0;
                    Parametrization.Inputs.AxisNo  := BYTE#1;
                    Parametrization.Inputs.HardwareId  := _AxisReference^.HWIDs.HW_ModuleAccessPoint;
                    IF AxisType = eAxoDriveAxisType#Rotary THEN
                        Parametrization.Inputs.ValueWriteLINT := TO_LINT(Position * -10000.0);
                    ELSIF AxisType = eAxoDriveAxisType#Linear THEN
                        Parametrization.Inputs.ValueWriteLINT := TO_LINT(Position * -10000000.0);
                    END_IF;
